	STP.B201B2_AirBlowerS2_RunStat AT %IX51.3 : BOOL;	(*  ~ {LinkedWith:TIID^C6920 (EtherCAT)^ScadaRoom_KouplerUTP (EK1100)^ScadaRoom_KouplerFiber (EK1521)^BlowerHouse_2 (EK1501)^Term 30 (EL1809)^Channel 14^Input} *)
	STP.B201B3_AirBlowerS2_RunStat AT %IX51.4 : BOOL;	(*  ~ {LinkedWith:TIID^C6920 (EtherCAT)^ScadaRoom_KouplerUTP (EK1100)^ScadaRoom_KouplerFiber (EK1521)^BlowerHouse_2 (EK1501)^Term 30 (EL1809)^Channel 15^Input} *)
	STP.M200B1A_MixerR1_LocalRemoteStat AT %IX51.5 : BOOL;	(*  ~ {LinkedWith:TIID^C6920 (EtherCAT)^ScadaRoom_KouplerUTP (EK1100)^ScadaRoom_KouplerFiber (EK1521)^BlowerHouse_2 (EK1501)^Term 31 (EL1809)^Channel 1^Input} *)
	STP.M200B1B_MixerR1_LocalRemoteStat AT %IX51.6 : BOOL;	(*  ~ {LinkedWith:TIID^C6920 (EtherCAT)^ScadaRoom_KouplerUTP (EK1100)^ScadaRoom_KouplerFiber (EK1521)^BlowerHouse_2 (EK1501)^Term 31 (EL1809)^Channel 2^Input} *)
	STP.M200B1C_MixerR1_LocalRemoteStat AT %IX51.7 : BOOL;	(*  ~ {LinkedWith:TIID^C6920 (EtherCAT)^ScadaRoom_KouplerUTP (EK1100)^ScadaRoom_KouplerFiber (EK1521)^BlowerHouse_2 (EK1501)^Term 31 (EL1809)^Channel 3^Input} *)
	STP.M200B2A_MixerR2_LocalRemoteStat AT %IX52.0 : BOOL;	(*  ~ {LinkedWith:TIID^C6920 (EtherCAT)^ScadaRoom_KouplerUTP (EK1100)^ScadaRoom_KouplerFiber (EK1521)^BlowerHouse_2 (EK1501)^Term 31 (EL1809)^Channel 4^Input} *)
	STP.M200B2B_MixerR2_LocalRemoteStat AT %IX52.1 : BOOL;	(*  ~ {LinkedWith:TIID^C6920 (EtherCAT)^ScadaRoom_KouplerUTP (EK1100)^ScadaRoom_KouplerFiber (EK1521)^BlowerHouse_2 (EK1501)^Term 31 (EL1809)^Channel 5^Input} *)
	STP.M200B2C_MixerR2_LocalRemoteStat AT %IX52.2 : BOOL;	(*  ~ {LinkedWith:TIID^C6920 (EtherCAT)^ScadaRoom_KouplerUTP (EK1100)^ScadaRoom_KouplerFiber (EK1521)^BlowerHouse_2 (EK1501)^Term 31 (EL1809)^Channel 6^Input} *)
	STP.M200B3A_MixerR3_LocalRemoteStat AT %IX52.3 : BOOL;	(*  ~ {LinkedWith:TIID^C6920 (EtherCAT)^ScadaRoom_KouplerUTP (EK1100)^ScadaRoom_KouplerFiber (EK1521)^BlowerHouse_2 (EK1501)^Term 31 (EL1809)^Channel 7^Input} *)
	STP.M200B3B_MixerR3_LocalRemoteStat AT %IX52.4 : BOOL;	(*  ~ {LinkedWith:TIID^C6920 (EtherCAT)^ScadaRoom_KouplerUTP (EK1100)^ScadaRoom_KouplerFiber (EK1521)^BlowerHouse_2 (EK1501)^Term 31 (EL1809)^Channel 8^Input} *)
	STP.M200B3C_MixerR3_LocalRemoteStat AT %IX52.5 : BOOL;	(*  ~ {LinkedWith:TIID^C6920 (EtherCAT)^ScadaRoom_KouplerUTP (EK1100)^ScadaRoom_KouplerFiber (EK1521)^BlowerHouse_2 (EK1501)^Term 31 (EL1809)^Channel 9^Input} *)
	STP.M200B4A_MixerR4_LocalRemoteStat AT %IX52.6 : BOOL;	(*  ~ {LinkedWith:TIID^C6920 (EtherCAT)^ScadaRoom_KouplerUTP (EK1100)^ScadaRoom_KouplerFiber (EK1521)^BlowerHouse_2 (EK1501)^Term 31 (EL1809)^Channel 10^Input} *)
	STP.M200B4B_MixerR4_LocalRemoteStat AT %IX52.7 : BOOL;	(*  ~ {LinkedWith:TIID^C6920 (EtherCAT)^ScadaRoom_KouplerUTP (EK1100)^ScadaRoom_KouplerFiber (EK1521)^BlowerHouse_2 (EK1501)^Term 31 (EL1809)^Channel 11^Input} *)
	STP.M200B4C_MixerR4_LocalRemoteStat AT %IX53.0 : BOOL;	(*  ~ {LinkedWith:TIID^C6920 (EtherCAT)^ScadaRoom_KouplerUTP (EK1100)^ScadaRoom_KouplerFiber (EK1521)^BlowerHouse_2 (EK1501)^Term 31 (EL1809)^Channel 12^Input} *)
	STP.B201B1_AirBlowerS2_LocalRemoteStat AT %IX53.1 : BOOL;	(*  ~ {LinkedWith:TIID^C6920 (EtherCAT)^ScadaRoom_KouplerUTP (EK1100)^ScadaRoom_KouplerFiber (EK1521)^BlowerHouse_2 (EK1501)^Term 32 (EL1809)^Channel 1^Input} *)
	STP.B201B2_AirBlowerS2_LocalRemoteStat AT %IX53.2 : BOOL;	(*  ~ {LinkedWith:TIID^C6920 (EtherCAT)^ScadaRoom_KouplerUTP (EK1100)^ScadaRoom_KouplerFiber (EK1521)^BlowerHouse_2 (EK1501)^Term 32 (EL1809)^Channel 2^Input} *)
	STP.B201B3_AirBlowerS2_LocalRemoteStat AT %IX53.3 : BOOL;	(*  ~ {LinkedWith:TIID^C6920 (EtherCAT)^ScadaRoom_KouplerUTP (EK1100)^ScadaRoom_KouplerFiber (EK1521)^BlowerHouse_2 (EK1501)^Term 32 (EL1809)^Channel 3^Input} *)
	STP.XV261B_DecanterR1_LocalRemoteStat AT %IX53.4 : BOOL;	(*  ~ {LinkedWith:TIID^C6920 (EtherCAT)^ScadaRoom_KouplerUTP (EK1100)^ScadaRoom_KouplerFiber (EK1521)^BlowerHouse_2 (EK1501)^Term 32 (EL1809)^Channel 4^Input} *)
	STP.XV262B_DecanterR2_LocalRemoteStat AT %IX53.5 : BOOL;	(*  ~ {LinkedWith:TIID^C6920 (EtherCAT)^ScadaRoom_KouplerUTP (EK1100)^ScadaRoom_KouplerFiber (EK1521)^BlowerHouse_2 (EK1501)^Term 32 (EL1809)^Channel 5^Input} *)
	STP.XV263B_DecanterR3_LocalRemoteStat AT %IX53.6 : BOOL;	(*  ~ {LinkedWith:TIID^C6920 (EtherCAT)^ScadaRoom_KouplerUTP (EK1100)^ScadaRoom_KouplerFiber (EK1521)^BlowerHouse_2 (EK1501)^Term 32 (EL1809)^Channel 6^Input} *)
	STP.XV264B_DecanterR4_LocalRemoteStat AT %IX53.7 : BOOL;	(*  ~ {LinkedWith:TIID^C6920 (EtherCAT)^ScadaRoom_KouplerUTP (EK1100)^ScadaRoom_KouplerFiber (EK1521)^BlowerHouse_2 (EK1501)^Term 32 (EL1809)^Channel 7^Input} *)
	STP.P201B1_DesludgePumpS2_LocalRemoteStat AT %IX54.0 : BOOL;	(*  ~ {LinkedWith:TIID^C6920 (EtherCAT)^ScadaRoom_KouplerUTP (EK1100)^ScadaRoom_KouplerFiber (EK1521)^BlowerHouse_2 (EK1501)^Term 32 (EL1809)^Channel 8^Input} *)
	STP.P201B2_DesludgePumpS2_LocalRemoteStat AT %IX54.1 : BOOL;	(*  ~ {LinkedWith:TIID^C6920 (EtherCAT)^ScadaRoom_KouplerUTP (EK1100)^ScadaRoom_KouplerFiber (EK1521)^BlowerHouse_2 (EK1501)^Term 32 (EL1809)^Channel 9^Input} *)
	STP.P201B1_DesludgePumpS2_RunStat AT %IX54.2 : BOOL;	(*  ~ {LinkedWith:TIID^C6920 (EtherCAT)^ScadaRoom_KouplerUTP (EK1100)^ScadaRoom_KouplerFiber (EK1521)^BlowerHouse_2 (EK1501)^Term 32 (EL1809)^Channel 10^Input} *)
	STP.P201B2_DesludgePumpS2_RunStat AT %IX54.3 : BOOL;	(*  ~ {LinkedWith:TIID^C6920 (EtherCAT)^ScadaRoom_KouplerUTP (EK1100)^ScadaRoom_KouplerFiber (EK1521)^BlowerHouse_2 (EK1501)^Term 32 (EL1809)^Channel 11^Input} *)
	STP.M200B1A_MixerR1_OverloadStat AT %IX54.4 : BOOL;	(*  ~ {LinkedWith:TIID^C6920 (EtherCAT)^ScadaRoom_KouplerUTP (EK1100)^ScadaRoom_KouplerFiber (EK1521)^BlowerHouse_2 (EK1501)^Term 33 (EL1809)^Channel 1^Input} *)
	STP.M200B1A_MixerR1_IncompleteStat AT %IX54.5 : BOOL;	(*  ~ {LinkedWith:TIID^C6920 (EtherCAT)^ScadaRoom_KouplerUTP (EK1100)^ScadaRoom_KouplerFiber (EK1521)^BlowerHouse_2 (EK1501)^Term 33 (EL1809)^Channel 2^Input} *)
	STP.M200B1B_MixerR1_OverloadStat AT %IX54.6 : BOOL;	(*  ~ {LinkedWith:TIID^C6920 (EtherCAT)^ScadaRoom_KouplerUTP (EK1100)^ScadaRoom_KouplerFiber (EK1521)^BlowerHouse_2 (EK1501)^Term 33 (EL1809)^Channel 3^Input} *)
	STP.M200B1B_MixerR1_IncompleteStat AT %IX54.7 : BOOL;	(*  ~ {LinkedWith:TIID^C6920 (EtherCAT)^ScadaRoom_KouplerUTP (EK1100)^ScadaRoom_KouplerFiber (EK1521)^BlowerHouse_2 (EK1501)^Term 33 (EL1809)^Channel 4^Input} *)
	STP.M200B1C_MixerR1_OverloadStat AT %IX55.0 : BOOL;	(*  ~ {LinkedWith:TIID^C6920 (EtherCAT)^ScadaRoom_KouplerUTP (EK1100)^ScadaRoom_KouplerFiber (EK1521)^BlowerHouse_2 (EK1501)^Term 33 (EL1809)^Channel 5^Input} *)
	STP.M200B1C_MixerR1_IncompleteStat AT %IX55.1 : BOOL;	(*  ~ {LinkedWith:TIID^C6920 (EtherCAT)^ScadaRoom_KouplerUTP (EK1100)^ScadaRoom_KouplerFiber (EK1521)^BlowerHouse_2 (EK1501)^Term 33 (EL1809)^Channel 6^Input} *)
	STP.M200B2A_MixerR2_OverloadStat AT %IX55.2 : BOOL;	(*  ~ {LinkedWith:TIID^C6920 (EtherCAT)^ScadaRoom_KouplerUTP (EK1100)^ScadaRoom_KouplerFiber (EK1521)^BlowerHouse_2 (EK1501)^Term 33 (EL1809)^Channel 7^Input} *)
	STP.M200B2A_MixerR2_IncompleteStat AT %IX55.3 : BOOL;	(*  ~ {LinkedWith:TIID^C6920 (EtherCAT)^ScadaRoom_KouplerUTP (EK1100)^ScadaRoom_KouplerFiber (EK1521)^BlowerHouse_2 (EK1501)^Term 33 (EL1809)^Channel 8^Input} *)
	STP.M200B2B_MixerR2_OverloadStat AT %IX55.4 : BOOL;	(*  ~ {LinkedWith:TIID^C6920 (EtherCAT)^ScadaRoom_KouplerUTP (EK1100)^ScadaRoom_KouplerFiber (EK1521)^BlowerHouse_2 (EK1501)^Term 33 (EL1809)^Channel 9^Input} *)
	STP.M200B2B_MixerR2_IncompleteStat AT %IX55.5 : BOOL;	(*  ~ {LinkedWith:TIID^C6920 (EtherCAT)^ScadaRoom_KouplerUTP (EK1100)^ScadaRoom_KouplerFiber (EK1521)^BlowerHouse_2 (EK1501)^Term 33 (EL1809)^Channel 10^Input} *)
	STP.M200B2C_MixerR2_OverloadStat AT %IX55.6 : BOOL;	(*  ~ {LinkedWith:TIID^C6920 (EtherCAT)^ScadaRoom_KouplerUTP (EK1100)^ScadaRoom_KouplerFiber (EK1521)^BlowerHouse_2 (EK1501)^Term 33 (EL1809)^Channel 11^Input} *)
	STP.M200B2C_MixerR2_IncompleteStat AT %IX55.7 : BOOL;	(*  ~ {LinkedWith:TIID^C6920 (EtherCAT)^ScadaRoom_KouplerUTP (EK1100)^ScadaRoom_KouplerFiber (EK1521)^BlowerHouse_2 (EK1501)^Term 33 (EL1809)^Channel 12^Input} *)
	STP.M200B3A_MixerR3_OverloadStat AT %IX56.0 : BOOL;	(*  ~ {LinkedWith:TIID^C6920 (EtherCAT)^ScadaRoom_KouplerUTP (EK1100)^ScadaRoom_KouplerFiber (EK1521)^BlowerHouse_2 (EK1501)^Term 33 (EL1809)^Channel 13^Input} *)
	STP.M200B3A_MixerR2_IncompleteStat AT %IX56.1 : BOOL;	(*  ~ {LinkedWith:TIID^C6920 (EtherCAT)^ScadaRoom_KouplerUTP (EK1100)^ScadaRoom_KouplerFiber (EK1521)^BlowerHouse_2 (EK1501)^Term 33 (EL1809)^Channel 14^Input} *)
	STP.M200B3B_MixerR3_OverloadStat AT %IX56.2 : BOOL;	(*  ~ {LinkedWith:TIID^C6920 (EtherCAT)^ScadaRoom_KouplerUTP (EK1100)^ScadaRoom_KouplerFiber (EK1521)^BlowerHouse_2 (EK1501)^Term 33 (EL1809)^Channel 15^Input} *)
	STP.M200B3B_MixerR3_IncompleteStat AT %IX56.3 : BOOL;	(*  ~ {LinkedWith:TIID^C6920 (EtherCAT)^ScadaRoom_KouplerUTP (EK1100)^ScadaRoom_KouplerFiber (EK1521)^BlowerHouse_2 (EK1501)^Term 33 (EL1809)^Channel 16^Input} *)
	STP.M200B3C_MixerR3_OverloadStat AT %IX56.4 : BOOL;	(*  ~ {LinkedWith:TIID^C6920 (EtherCAT)^ScadaRoom_KouplerUTP (EK1100)^ScadaRoom_KouplerFiber (EK1521)^BlowerHouse_2 (EK1501)^Term 34 (EL1809)^Channel 1^Input} *)
	STP.M200B3C_MixerR3_IncompleteStat AT %IX56.5 : BOOL;	(*  ~ {LinkedWith:TIID^C6920 (EtherCAT)^ScadaRoom_KouplerUTP (EK1100)^ScadaRoom_KouplerFiber (EK1521)^BlowerHouse_2 (EK1501)^Term 34 (EL1809)^Channel 2^Input} *)
	STP.M200B4A_MixerR4_OverloadStat AT %IX56.6 : BOOL;	(*  ~ {LinkedWith:TIID^C6920 (EtherCAT)^ScadaRoom_KouplerUTP (EK1100)^ScadaRoom_KouplerFiber (EK1521)^BlowerHouse_2 (EK1501)^Term 34 (EL1809)^Channel 3^Input} *)
	STP.M200B4A_MixerR4_IncompleteStat AT %IX56.7 : BOOL;	(*  ~ {LinkedWith:TIID^C6920 (EtherCAT)^ScadaRoom_KouplerUTP (EK1100)^ScadaRoom_KouplerFiber (EK1521)^BlowerHouse_2 (EK1501)^Term 34 (EL1809)^Channel 4^Input} *)
	STP.M200B4B_MixerR4_OverloadStat AT %IX257.0 : BOOL;	(*  ~ {LinkedWith:TIID^C6920 (EtherCAT)^ScadaRoom_KouplerUTP (EK1100)^ScadaRoom_KouplerFiber (EK1521)^BlowerHouse_2 (EK1501)^Term 34 (EL1809)^Channel 5^Input} *)
	STP.M200B4B_MixerR4_IncompleteStat AT %IX57.0 : BOOL;	(*  ~ {LinkedWith:TIID^C6920 (EtherCAT)^ScadaRoom_KouplerUTP (EK1100)^ScadaRoom_KouplerFiber (EK1521)^BlowerHouse_2 (EK1501)^Term 34 (EL1809)^Channel 6^Input} *)
	STP.M200B4C_MixerR4_OverloadStat AT %IX57.1 : BOOL;	(*  ~ {LinkedWith:TIID^C6920 (EtherCAT)^ScadaRoom_KouplerUTP (EK1100)^ScadaRoom_KouplerFiber (EK1521)^BlowerHouse_2 (EK1501)^Term 34 (EL1809)^Channel 7^Input} *)
	STP.M200B4C_MixerR4_IncompleteStat AT %IX57.2 : BOOL;	(*  ~ {LinkedWith:TIID^C6920 (EtherCAT)^ScadaRoom_KouplerUTP (EK1100)^ScadaRoom_KouplerFiber (EK1521)^BlowerHouse_2 (EK1501)^Term 34 (EL1809)^Channel 8^Input} *)
	STP.B201B1_AirBlowerS2_OverloadStat AT %IX57.3 : BOOL;	(*  ~ {LinkedWith:TIID^C6920 (EtherCAT)^ScadaRoom_KouplerUTP (EK1100)^ScadaRoom_KouplerFiber (EK1521)^BlowerHouse_2 (EK1501)^Term 34 (EL1809)^Channel 9^Input} *)
	STP.B201B1_AirBlowerS2_IncompleteStat AT %IX57.4 : BOOL;	(*  ~ {LinkedWith:TIID^C6920 (EtherCAT)^ScadaRoom_KouplerUTP (EK1100)^ScadaRoom_KouplerFiber (EK1521)^BlowerHouse_2 (EK1501)^Term 34 (EL1809)^Channel 10^Input} *)
	STP.B201B2_AirBlowerS2_OverloadStat AT %IX57.5 : BOOL;	(*  ~ {LinkedWith:TIID^C6920 (EtherCAT)^ScadaRoom_KouplerUTP (EK1100)^ScadaRoom_KouplerFiber (EK1521)^BlowerHouse_2 (EK1501)^Term 34 (EL1809)^Channel 11^Input} *)
	STP.B201B2_AirBlowerS2_IncompleteStat AT %IX57.6 : BOOL;	(*  ~ {LinkedWith:TIID^C6920 (EtherCAT)^ScadaRoom_KouplerUTP (EK1100)^ScadaRoom_KouplerFiber (EK1521)^BlowerHouse_2 (EK1501)^Term 34 (EL1809)^Channel 12^Input} *)
	STP.B201B3_AirBlowerS2_OverloadStat AT %IX57.7 : BOOL;	(*  ~ {LinkedWith:TIID^C6920 (EtherCAT)^ScadaRoom_KouplerUTP (EK1100)^ScadaRoom_KouplerFiber (EK1521)^BlowerHouse_2 (EK1501)^Term 34 (EL1809)^Channel 13^Input} *)
	STP.B201B3_AirBlowerS2_IncompleteStat AT %IX58.0 : BOOL;	(*  ~ {LinkedWith:TIID^C6920 (EtherCAT)^ScadaRoom_KouplerUTP (EK1100)^ScadaRoom_KouplerFiber (EK1521)^BlowerHouse_2 (EK1501)^Term 34 (EL1809)^Channel 14^Input} *)
	STP.P201B1_DesludgePumpS2_OverloadStat AT %IX58.1 : BOOL;	(*  ~ {LinkedWith:TIID^C6920 (EtherCAT)^ScadaRoom_KouplerUTP (EK1100)^ScadaRoom_KouplerFiber (EK1521)^BlowerHouse_2 (EK1501)^Term 34 (EL1809)^Channel 15^Input} *)
	STP.P201B2_DesludgePumpS2_OverloadStat AT %IX58.2 : BOOL;	(*  ~ {LinkedWith:TIID^C6920 (EtherCAT)^ScadaRoom_KouplerUTP (EK1100)^ScadaRoom_KouplerFiber (EK1521)^BlowerHouse_2 (EK1501)^Term 34 (EL1809)^Channel 16^Input} *)
	STP.M200B1A_MixerR1_EStopStat AT %IX58.3 : BOOL;	(*  ~ {LinkedWith:TIID^C6920 (EtherCAT)^ScadaRoom_KouplerUTP (EK1100)^ScadaRoom_KouplerFiber (EK1521)^BlowerHouse_2 (EK1501)^Term 35 (EL1809)^Channel 1^Input} *)
	STP.M200B1B_MixerR1_EStopStat AT %IX58.4 : BOOL;	(*  ~ {LinkedWith:TIID^C6920 (EtherCAT)^ScadaRoom_KouplerUTP (EK1100)^ScadaRoom_KouplerFiber (EK1521)^BlowerHouse_2 (EK1501)^Term 35 (EL1809)^Channel 2^Input} *)
	STP.M200B1C_MixerR1_EStopStat AT %IX58.5 : BOOL;	(*  ~ {LinkedWith:TIID^C6920 (EtherCAT)^ScadaRoom_KouplerUTP (EK1100)^ScadaRoom_KouplerFiber (EK1521)^BlowerHouse_2 (EK1501)^Term 35 (EL1809)^Channel 3^Input} *)
	STP.M200B2A_MixerR2_EStopStat AT %IX58.6 : BOOL;	(*  ~ {LinkedWith:TIID^C6920 (EtherCAT)^ScadaRoom_KouplerUTP (EK1100)^ScadaRoom_KouplerFiber (EK1521)^BlowerHouse_2 (EK1501)^Term 35 (EL1809)^Channel 4^Input} *)
	STP.M200B2B_MixerR2_EStopStat AT %IX58.7 : BOOL;	(*  ~ {LinkedWith:TIID^C6920 (EtherCAT)^ScadaRoom_KouplerUTP (EK1100)^ScadaRoom_KouplerFiber (EK1521)^BlowerHouse_2 (EK1501)^Term 35 (EL1809)^Channel 5^Input} *)
	STP.M200B2C_MixerR2_EStopStat AT %IX59.0 : BOOL;	(*  ~ {LinkedWith:TIID^C6920 (EtherCAT)^ScadaRoom_KouplerUTP (EK1100)^ScadaRoom_KouplerFiber (EK1521)^BlowerHouse_2 (EK1501)^Term 35 (EL1809)^Channel 6^Input} *)
	STP.M200B3A_MixerR3_EStopStat AT %IX59.1 : BOOL;	(*  ~ {LinkedWith:TIID^C6920 (EtherCAT)^ScadaRoom_KouplerUTP (EK1100)^ScadaRoom_KouplerFiber (EK1521)^BlowerHouse_2 (EK1501)^Term 35 (EL1809)^Channel 7^Input} *)
	STP.M200B3B_MixerR3_EStopStat AT %IX59.2 : BOOL;	(*  ~ {LinkedWith:TIID^C6920 (EtherCAT)^ScadaRoom_KouplerUTP (EK1100)^ScadaRoom_KouplerFiber (EK1521)^BlowerHouse_2 (EK1501)^Term 35 (EL1809)^Channel 8^Input} *)
	STP.M200B3C_MixerR3_EStopStat AT %IX59.3 : BOOL;	(*  ~ {LinkedWith:TIID^C6920 (EtherCAT)^ScadaRoom_KouplerUTP (EK1100)^ScadaRoom_KouplerFiber (EK1521)^BlowerHouse_2 (EK1501)^Term 35 (EL1809)^Channel 9^Input} *)
	STP.M200B4A_MixerR4_EStopStat AT %IX59.4 : BOOL;	(*  ~ {LinkedWith:TIID^C6920 (EtherCAT)^ScadaRoom_KouplerUTP (EK1100)^ScadaRoom_KouplerFiber (EK1521)^BlowerHouse_2 (EK1501)^Term 35 (EL1809)^Channel 10^Input} *)
	STP.M200B4B_MixerR4_EStopStat AT %IX59.5 : BOOL;	(*  ~ {LinkedWith:TIID^C6920 (EtherCAT)^ScadaRoom_KouplerUTP (EK1100)^ScadaRoom_KouplerFiber (EK1521)^BlowerHouse_2 (EK1501)^Term 35 (EL1809)^Channel 11^Input} *)
	STP.M200B4C_MixerR4_EStopStat AT %IX59.6 : BOOL;	(*  ~ {LinkedWith:TIID^C6920 (EtherCAT)^ScadaRoom_KouplerUTP (EK1100)^ScadaRoom_KouplerFiber (EK1521)^BlowerHouse_2 (EK1501)^Term 35 (EL1809)^Channel 12^Input} *)
	STP.B201B1_AirBlowerS2_EStopStat AT %IX59.7 : BOOL;	(*  ~ {LinkedWith:TIID^C6920 (EtherCAT)^ScadaRoom_KouplerUTP (EK1100)^ScadaRoom_KouplerFiber (EK1521)^BlowerHouse_2 (EK1501)^Term 36 (EL1809)^Channel 1^Input} *)
	STP.B201B2_AirBlowerS2_EStopStat AT %IX60.0 : BOOL;	(*  ~ {LinkedWith:TIID^C6920 (EtherCAT)^ScadaRoom_KouplerUTP (EK1100)^ScadaRoom_KouplerFiber (EK1521)^BlowerHouse_2 (EK1501)^Term 36 (EL1809)^Channel 2^Input} *)
	STP.B201B3_AirBlowerS2_EStopStat AT %IX60.1 : BOOL;	(*  ~ {LinkedWith:TIID^C6920 (EtherCAT)^ScadaRoom_KouplerUTP (EK1100)^ScadaRoom_KouplerFiber (EK1521)^BlowerHouse_2 (EK1501)^Term 36 (EL1809)^Channel 3^Input} *)
	STP.XV261B_DecanterR1_EStopStat AT %IX60.2 : BOOL;	(*  ~ {LinkedWith:TIID^C6920 (EtherCAT)^ScadaRoom_KouplerUTP (EK1100)^ScadaRoom_KouplerFiber (EK1521)^BlowerHouse_2 (EK1501)^Term 36 (EL1809)^Channel 4^Input} *)
	STP.XV262B_DecanterR2_EStopStat AT %IX60.3 : BOOL;	(*  ~ {LinkedWith:TIID^C6920 (EtherCAT)^ScadaRoom_KouplerUTP (EK1100)^ScadaRoom_KouplerFiber (EK1521)^BlowerHouse_2 (EK1501)^Term 36 (EL1809)^Channel 5^Input} *)
	STP.XV263B_DecanterR3_EStopStat AT %IX60.4 : BOOL;	(*  ~ {LinkedWith:TIID^C6920 (EtherCAT)^ScadaRoom_KouplerUTP (EK1100)^ScadaRoom_KouplerFiber (EK1521)^BlowerHouse_2 (EK1501)^Term 36 (EL1809)^Channel 6^Input} *)
	STP.XV264B_DecanterR4_EStopStat AT %IX60.5 : BOOL;	(*  ~ {LinkedWith:TIID^C6920 (EtherCAT)^ScadaRoom_KouplerUTP (EK1100)^ScadaRoom_KouplerFiber (EK1521)^BlowerHouse_2 (EK1501)^Term 36 (EL1809)^Channel 7^Input} *)
	STP.P201B1_DesludgePumpS2_EStopStat AT %IX60.6 : BOOL;	(*  ~ {LinkedWith:TIID^C6920 (EtherCAT)^ScadaRoom_KouplerUTP (EK1100)^ScadaRoom_KouplerFiber (EK1521)^BlowerHouse_2 (EK1501)^Term 36 (EL1809)^Channel 8^Input} *)
	STP.P201B2_DesludgePumpS2_EStopStat AT %IX60.7 : BOOL;	(*  ~ {LinkedWith:TIID^C6920 (EtherCAT)^ScadaRoom_KouplerUTP (EK1100)^ScadaRoom_KouplerFiber (EK1521)^BlowerHouse_2 (EK1501)^Term 36 (EL1809)^Channel 9^Input} *)
	STP.XV261B_DecanterR1_FwdStat AT %IX61.0 : BOOL;	(*  ~ {LinkedWith:TIID^C6920 (EtherCAT)^ScadaRoom_KouplerUTP (EK1100)^ScadaRoom_KouplerFiber (EK1521)^BlowerHouse_2 (EK1501)^Term 37 (EL1809)^Channel 1^Input} *)
	STP.XV262B_DecanterR2_FwdStat AT %IX61.1 : BOOL;	(*  ~ {LinkedWith:TIID^C6920 (EtherCAT)^ScadaRoom_KouplerUTP (EK1100)^ScadaRoom_KouplerFiber (EK1521)^BlowerHouse_2 (EK1501)^Term 37 (EL1809)^Channel 2^Input} *)
	STP.XV263B_DecanterR3_FwdStat AT %IX61.2 : BOOL;	(*  ~ {LinkedWith:TIID^C6920 (EtherCAT)^ScadaRoom_KouplerUTP (EK1100)^ScadaRoom_KouplerFiber (EK1521)^BlowerHouse_2 (EK1501)^Term 37 (EL1809)^Channel 3^Input} *)
	STP.XV264B_DecanterR4_FwdStat AT %IX61.3 : BOOL;	(*  ~ {LinkedWith:TIID^C6920 (EtherCAT)^ScadaRoom_KouplerUTP (EK1100)^ScadaRoom_KouplerFiber (EK1521)^BlowerHouse_2 (EK1501)^Term 37 (EL1809)^Channel 4^Input} *)
	STP.XV261B_DecanterR1_RvsStat AT %IX61.4 : BOOL;	(*  ~ {LinkedWith:TIID^C6920 (EtherCAT)^ScadaRoom_KouplerUTP (EK1100)^ScadaRoom_KouplerFiber (EK1521)^BlowerHouse_2 (EK1501)^Term 37 (EL1809)^Channel 5^Input} *)
	STP.XV262B_DecanterR2_RvsStat AT %IX61.5 : BOOL;	(*  ~ {LinkedWith:TIID^C6920 (EtherCAT)^ScadaRoom_KouplerUTP (EK1100)^ScadaRoom_KouplerFiber (EK1521)^BlowerHouse_2 (EK1501)^Term 37 (EL1809)^Channel 6^Input} *)
	STP.XV263B_DecanterR3_RvsStat AT %IX61.6 : BOOL;	(*  ~ {LinkedWith:TIID^C6920 (EtherCAT)^ScadaRoom_KouplerUTP (EK1100)^ScadaRoom_KouplerFiber (EK1521)^BlowerHouse_2 (EK1501)^Term 37 (EL1809)^Channel 7^Input} *)
	STP.XV264B_DecanterR4_RvsStat AT %IX61.7 : BOOL;	(*  ~ {LinkedWith:TIID^C6920 (EtherCAT)^ScadaRoom_KouplerUTP (EK1100)^ScadaRoom_KouplerFiber (EK1521)^BlowerHouse_2 (EK1501)^Term 37 (EL1809)^Channel 8^Input} *)
	STP.M200B1A_MixerR1_RunCmd AT %QX17.1 : BOOL;	(*  ~ {LinkedWith:TIID^C6920 (EtherCAT)^ScadaRoom_KouplerUTP (EK1100)^ScadaRoom_KouplerFiber (EK1521)^BlowerHouse_2 (EK1501)^Term 39 (EL2809)^Channel 1^Output} *)
	STP.M200B1B_MixerR1_RunCmd AT %QX17.2 : BOOL;	(*  ~ {LinkedWith:TIID^C6920 (EtherCAT)^ScadaRoom_KouplerUTP (EK1100)^ScadaRoom_KouplerFiber (EK1521)^BlowerHouse_2 (EK1501)^Term 39 (EL2809)^Channel 2^Output} *)
	STP.M200B1C_MixerR1_RunCmd AT %QX17.3 : BOOL;	(*  ~ {LinkedWith:TIID^C6920 (EtherCAT)^ScadaRoom_KouplerUTP (EK1100)^ScadaRoom_KouplerFiber (EK1521)^BlowerHouse_2 (EK1501)^Term 39 (EL2809)^Channel 3^Output} *)
	STP.M200B2A_MixerR2_RunCmd AT %QX17.4 : BOOL;	(*  ~ {LinkedWith:TIID^C6920 (EtherCAT)^ScadaRoom_KouplerUTP (EK1100)^ScadaRoom_KouplerFiber (EK1521)^BlowerHouse_2 (EK1501)^Term 39 (EL2809)^Channel 4^Output} *)
	STP.M200B2B_MixerR2_RunCmd AT %QX17.5 : BOOL;	(*  ~ {LinkedWith:TIID^C6920 (EtherCAT)^ScadaRoom_KouplerUTP (EK1100)^ScadaRoom_KouplerFiber (EK1521)^BlowerHouse_2 (EK1501)^Term 39 (EL2809)^Channel 5^Output} *)
	STP.M200B2C_MixerR2_RunCmd AT %QX17.6 : BOOL;	(*  ~ {LinkedWith:TIID^C6920 (EtherCAT)^ScadaRoom_KouplerUTP (EK1100)^ScadaRoom_KouplerFiber (EK1521)^BlowerHouse_2 (EK1501)^Term 39 (EL2809)^Channel 6^Output} *)
	STP.M200B3A_MixerR3_RunCmd AT %QX17.7 : BOOL;	(*  ~ {LinkedWith:TIID^C6920 (EtherCAT)^ScadaRoom_KouplerUTP (EK1100)^ScadaRoom_KouplerFiber (EK1521)^BlowerHouse_2 (EK1501)^Term 39 (EL2809)^Channel 7^Output} *)
	STP.M200B3B_MixerR3_RunCmd AT %QX18.0 : BOOL;	(*  ~ {LinkedWith:TIID^C6920 (EtherCAT)^ScadaRoom_KouplerUTP (EK1100)^ScadaRoom_KouplerFiber (EK1521)^BlowerHouse_2 (EK1501)^Term 39 (EL2809)^Channel 8^Output} *)
	STP.M200B3C_MixerR3_RunCmd AT %QX18.1 : BOOL;	(*  ~ {LinkedWith:TIID^C6920 (EtherCAT)^ScadaRoom_KouplerUTP (EK1100)^ScadaRoom_KouplerFiber (EK1521)^BlowerHouse_2 (EK1501)^Term 39 (EL2809)^Channel 9^Output} *)
	STP.M200B4A_MixerR4_RunCmd AT %QX18.2 : BOOL;	(*  ~ {LinkedWith:TIID^C6920 (EtherCAT)^ScadaRoom_KouplerUTP (EK1100)^ScadaRoom_KouplerFiber (EK1521)^BlowerHouse_2 (EK1501)^Term 39 (EL2809)^Channel 10^Output} *)
	STP.M200B4B_MixerR4_RunCmd AT %QX18.3 : BOOL;	(*  ~ {LinkedWith:TIID^C6920 (EtherCAT)^ScadaRoom_KouplerUTP (EK1100)^ScadaRoom_KouplerFiber (EK1521)^BlowerHouse_2 (EK1501)^Term 39 (EL2809)^Channel 11^Output} *)
	STP.M200B4C_MixerR4_RunCmd AT %QX18.4 : BOOL;	(*  ~ {LinkedWith:TIID^C6920 (EtherCAT)^ScadaRoom_KouplerUTP (EK1100)^ScadaRoom_KouplerFiber (EK1521)^BlowerHouse_2 (EK1501)^Term 39 (EL2809)^Channel 12^Output} *)
	STP.XV261B_DecanterR1_FwdCmd AT %QX18.5 : BOOL;	(*  ~ {LinkedWith:TIID^C6920 (EtherCAT)^ScadaRoom_KouplerUTP (EK1100)^ScadaRoom_KouplerFiber (EK1521)^BlowerHouse_2 (EK1501)^Term 40 (EL2809)^Channel 1^Output} *)
	STP.XV262B_DecanterR2_FwdCmd AT %QX18.6 : BOOL;	(*  ~ {LinkedWith:TIID^C6920 (EtherCAT)^ScadaRoom_KouplerUTP (EK1100)^ScadaRoom_KouplerFiber (EK1521)^BlowerHouse_2 (EK1501)^Term 40 (EL2809)^Channel 2^Output} *)
	STP.XV263B_DecanterR3_FwdCmd AT %QX18.7 : BOOL;	(*  ~ {LinkedWith:TIID^C6920 (EtherCAT)^ScadaRoom_KouplerUTP (EK1100)^ScadaRoom_KouplerFiber (EK1521)^BlowerHouse_2 (EK1501)^Term 40 (EL2809)^Channel 3^Output} *)
	STP.XV264B_DecanterR4_FwdCmd AT %QX19.0 : BOOL;	(*  ~ {LinkedWith:TIID^C6920 (EtherCAT)^ScadaRoom_KouplerUTP (EK1100)^ScadaRoom_KouplerFiber (EK1521)^BlowerHouse_2 (EK1501)^Term 40 (EL2809)^Channel 4^Output} *)
	STP.XV261B_DecanterR1_RvsCmd AT %QX19.1 : BOOL;	(*  ~ {LinkedWith:TIID^C6920 (EtherCAT)^ScadaRoom_KouplerUTP (EK1100)^ScadaRoom_KouplerFiber (EK1521)^BlowerHouse_2 (EK1501)^Term 40 (EL2809)^Channel 5^Output} *)
	STP.XV262B_DecanterR2_RvsCmd AT %QX19.2 : BOOL;	(*  ~ {LinkedWith:TIID^C6920 (EtherCAT)^ScadaRoom_KouplerUTP (EK1100)^ScadaRoom_KouplerFiber (EK1521)^BlowerHouse_2 (EK1501)^Term 40 (EL2809)^Channel 6^Output} *)
	STP.XV263B_DecanterR3_RvsCmd AT %QX19.3 : BOOL;	(*  ~ {LinkedWith:TIID^C6920 (EtherCAT)^ScadaRoom_KouplerUTP (EK1100)^ScadaRoom_KouplerFiber (EK1521)^BlowerHouse_2 (EK1501)^Term 40 (EL2809)^Channel 7^Output} *)
	STP.XV264B_DecanterR4_RvsCmd AT %QX19.4 : BOOL;	(*  ~ {LinkedWith:TIID^C6920 (EtherCAT)^ScadaRoom_KouplerUTP (EK1100)^ScadaRoom_KouplerFiber (EK1521)^BlowerHouse_2 (EK1501)^Term 40 (EL2809)^Channel 8^Output} *)
	STP.B201B1_AirBlowerS2_RunCmd AT %QX19.5 : BOOL;	(*  ~ {LinkedWith:TIID^C6920 (EtherCAT)^ScadaRoom_KouplerUTP (EK1100)^ScadaRoom_KouplerFiber (EK1521)^BlowerHouse_2 (EK1501)^Term 40 (EL2809)^Channel 9^Output} *)
	STP.B201B2_AirBlowerS2_RunCmd AT %QX19.6 : BOOL;	(*  ~ {LinkedWith:TIID^C6920 (EtherCAT)^ScadaRoom_KouplerUTP (EK1100)^ScadaRoom_KouplerFiber (EK1521)^BlowerHouse_2 (EK1501)^Term 40 (EL2809)^Channel 10^Output} *)
	STP.B201B3_AirBlowerS2_RunCmd AT %QX19.7 : BOOL;	(*  ~ {LinkedWith:TIID^C6920 (EtherCAT)^ScadaRoom_KouplerUTP (EK1100)^ScadaRoom_KouplerFiber (EK1521)^BlowerHouse_2 (EK1501)^Term 40 (EL2809)^Channel 11^Output} *)
	STP.P201B1_DesludgePumpS2_RunCmd AT %QX20.0 : BOOL;	(*  ~ {LinkedWith:TIID^C6920 (EtherCAT)^ScadaRoom_KouplerUTP (EK1100)^ScadaRoom_KouplerFiber (EK1521)^BlowerHouse_2 (EK1501)^Term 40 (EL2809)^Channel 12^Output} *)
	STP.P201B2_DesludgePumpS2_RunCmd AT %QX20.1 : BOOL;	(*  ~ {LinkedWith:TIID^C6920 (EtherCAT)^ScadaRoom_KouplerUTP (EK1100)^ScadaRoom_KouplerFiber (EK1521)^BlowerHouse_2 (EK1501)^Term 40 (EL2809)^Channel 13^Output} *)
	STP.LSH201A1_LevelSensorR1 AT %IX64.0 : BOOL;	(*  ~ {LinkedWith:TIID^C6920 (EtherCAT)^ScadaRoom_KouplerUTP (EK1100)^ScadaRoom_KouplerFiber (EK1521)^SBR_1 (EK1501)^Term 57 (EL1809)^Channel 1^Input} *)
	STP.LSH201A2_LevelSensorR2 AT %IX64.1 : BOOL;	(*  ~ {LinkedWith:TIID^C6920 (EtherCAT)^ScadaRoom_KouplerUTP (EK1100)^ScadaRoom_KouplerFiber (EK1521)^SBR_1 (EK1501)^Term 57 (EL1809)^Channel 2^Input} *)
	STP.LSH201A3_LevelSensorR3 AT %IX64.2 : BOOL;	(*  ~ {LinkedWith:TIID^C6920 (EtherCAT)^ScadaRoom_KouplerUTP (EK1100)^ScadaRoom_KouplerFiber (EK1521)^SBR_1 (EK1501)^Term 57 (EL1809)^Channel 3^Input} *)
	STP.LSH201A4_LevelSensorR4 AT %IX64.3 : BOOL;	(*  ~ {LinkedWith:TIID^C6920 (EtherCAT)^ScadaRoom_KouplerUTP (EK1100)^ScadaRoom_KouplerFiber (EK1521)^SBR_1 (EK1501)^Term 57 (EL1809)^Channel 4^Input} *)
	STP.OPR1A_ReactorStatus AT %IX64.4 : BOOL;	(*  ~ {LinkedWith:TIID^C6920 (EtherCAT)^ScadaRoom_KouplerUTP (EK1100)^ScadaRoom_KouplerFiber (EK1521)^SBR_1 (EK1501)^Term 57 (EL1809)^Channel 5^Input} *)
	STP.OPR2A_ReactorStatus AT %IX64.5 : BOOL;	(*  ~ {LinkedWith:TIID^C6920 (EtherCAT)^ScadaRoom_KouplerUTP (EK1100)^ScadaRoom_KouplerFiber (EK1521)^SBR_1 (EK1501)^Term 57 (EL1809)^Channel 6^Input} *)
	STP.OPR3A_ReactorStatus AT %IX64.6 : BOOL;	(*  ~ {LinkedWith:TIID^C6920 (EtherCAT)^ScadaRoom_KouplerUTP (EK1100)^ScadaRoom_KouplerFiber (EK1521)^SBR_1 (EK1501)^Term 57 (EL1809)^Channel 7^Input} *)
	STP.OPR4A_ReactorStatus AT %IX64.7 : BOOL;	(*  ~ {LinkedWith:TIID^C6920 (EtherCAT)^ScadaRoom_KouplerUTP (EK1100)^ScadaRoom_KouplerFiber (EK1521)^SBR_1 (EK1501)^Term 57 (EL1809)^Channel 8^Input} *)
	STP.DP04_DoorPanelStatus AT %IX65.0 : BOOL;	(*  ~ {LinkedWith:TIID^C6920 (EtherCAT)^ScadaRoom_KouplerUTP (EK1100)^ScadaRoom_KouplerFiber (EK1521)^SBR_1 (EK1501)^Term 57 (EL1809)^Channel 9^Input} *)
	STP.TMT04_FanStatus AT %IX65.1 : BOOL;	(*  ~ {LinkedWith:TIID^C6920 (EtherCAT)^ScadaRoom_KouplerUTP (EK1100)^ScadaRoom_KouplerFiber (EK1521)^SBR_1 (EK1501)^Term 57 (EL1809)^Channel 10^Input} *)
	STP.HR201A1_DecantHighLevelR1 AT %IX65.2 : BOOL;	(*  ~ {LinkedWith:TIID^C6920 (EtherCAT)^ScadaRoom_KouplerUTP (EK1100)^ScadaRoom_KouplerFiber (EK1521)^SBR_1 (EK1501)^Term 58 (EL1809)^Channel 1^Input} *)
	STP.LR201A1_DecantLowLevelR1 AT %IX65.3 : BOOL;	(*  ~ {LinkedWith:TIID^C6920 (EtherCAT)^ScadaRoom_KouplerUTP (EK1100)^ScadaRoom_KouplerFiber (EK1521)^SBR_1 (EK1501)^Term 58 (EL1809)^Channel 2^Input} *)
	STP.HR201A2_DecantHighLevelR2 AT %IX65.4 : BOOL;	(*  ~ {LinkedWith:TIID^C6920 (EtherCAT)^ScadaRoom_KouplerUTP (EK1100)^ScadaRoom_KouplerFiber (EK1521)^SBR_1 (EK1501)^Term 58 (EL1809)^Channel 3^Input} *)
	STP.LR201A2_DecantLowLevelR2 AT %IX65.5 : BOOL;	(*  ~ {LinkedWith:TIID^C6920 (EtherCAT)^ScadaRoom_KouplerUTP (EK1100)^ScadaRoom_KouplerFiber (EK1521)^SBR_1 (EK1501)^Term 58 (EL1809)^Channel 4^Input} *)
	STP.HR201A3_DecantHighLevelR3 AT %IX65.6 : BOOL;	(*  ~ {LinkedWith:TIID^C6920 (EtherCAT)^ScadaRoom_KouplerUTP (EK1100)^ScadaRoom_KouplerFiber (EK1521)^SBR_1 (EK1501)^Term 58 (EL1809)^Channel 5^Input} *)
	STP.LR201A3_DecantLowLevelR3 AT %IX65.7 : BOOL;	(*  ~ {LinkedWith:TIID^C6920 (EtherCAT)^ScadaRoom_KouplerUTP (EK1100)^ScadaRoom_KouplerFiber (EK1521)^SBR_1 (EK1501)^Term 58 (EL1809)^Channel 6^Input} *)
	STP.HR201A4_DecantHighLevelR4 AT %IX66.0 : BOOL;	(*  ~ {LinkedWith:TIID^C6920 (EtherCAT)^ScadaRoom_KouplerUTP (EK1100)^ScadaRoom_KouplerFiber (EK1521)^SBR_1 (EK1501)^Term 58 (EL1809)^Channel 7^Input} *)
	STP.LR201A4_DecantLowLevelR4 AT %IX66.1 : BOOL;	(*  ~ {LinkedWith:TIID^C6920 (EtherCAT)^ScadaRoom_KouplerUTP (EK1100)^ScadaRoom_KouplerFiber (EK1521)^SBR_1 (EK1501)^Term 58 (EL1809)^Channel 8^Input} *)
	STP.XV205A_SBRValveR1_OpenStat AT %IX66.2 : BOOL;	(*  ~ {LinkedWith:TIID^C6920 (EtherCAT)^ScadaRoom_KouplerUTP (EK1100)^ScadaRoom_KouplerFiber (EK1521)^SBR_1 (EK1501)^Term 59 (EL1809)^Channel 1^Input} *)
	STP.XV206A_SBRValveR2_OpenStat AT %IX66.3 : BOOL;	(*  ~ {LinkedWith:TIID^C6920 (EtherCAT)^ScadaRoom_KouplerUTP (EK1100)^ScadaRoom_KouplerFiber (EK1521)^SBR_1 (EK1501)^Term 59 (EL1809)^Channel 2^Input} *)
	STP.XV207A_SBRValveR3_OpenStat AT %IX66.4 : BOOL;	(*  ~ {LinkedWith:TIID^C6920 (EtherCAT)^ScadaRoom_KouplerUTP (EK1100)^ScadaRoom_KouplerFiber (EK1521)^SBR_1 (EK1501)^Term 59 (EL1809)^Channel 3^Input} *)
	STP.XV208A_SBRValveR4_OpenStat AT %IX66.5 : BOOL;	(*  ~ {LinkedWith:TIID^C6920 (EtherCAT)^ScadaRoom_KouplerUTP (EK1100)^ScadaRoom_KouplerFiber (EK1521)^SBR_1 (EK1501)^Term 59 (EL1809)^Channel 4^Input} *)
	STP.XV201A_AirBlowerValveR1_OpenStat AT %IX66.6 : BOOL;	(*  ~ {LinkedWith:TIID^C6920 (EtherCAT)^ScadaRoom_KouplerUTP (EK1100)^ScadaRoom_KouplerFiber (EK1521)^SBR_1 (EK1501)^Term 59 (EL1809)^Channel 5^Input} *)
	STP.XV202A_AirBlowerValveR2_OpenStat AT %IX66.7 : BOOL;	(*  ~ {LinkedWith:TIID^C6920 (EtherCAT)^ScadaRoom_KouplerUTP (EK1100)^ScadaRoom_KouplerFiber (EK1521)^SBR_1 (EK1501)^Term 59 (EL1809)^Channel 6^Input} *)
	STP.XV203A_AirBlowerValveR3_OpenStat AT %IX67.0 : BOOL;	(*  ~ {LinkedWith:TIID^C6920 (EtherCAT)^ScadaRoom_KouplerUTP (EK1100)^ScadaRoom_KouplerFiber (EK1521)^SBR_1 (EK1501)^Term 59 (EL1809)^Channel 7^Input} *)
	STP.XV204A_AirBlowerValveR4_OpenStat AT %IX68.1 : BOOL;	(*  ~ {LinkedWith:TIID^C6920 (EtherCAT)^ScadaRoom_KouplerUTP (EK1100)^ScadaRoom_KouplerFiber (EK1521)^SBR_1 (EK1501)^Term 59 (EL1809)^Channel 8^Input} *)
	STP.XV221A_LimeValveR1_OpenStat AT %IX67.1 : BOOL;	(*  ~ {LinkedWith:TIID^C6920 (EtherCAT)^ScadaRoom_KouplerUTP (EK1100)^ScadaRoom_KouplerFiber (EK1521)^SBR_1 (EK1501)^Term 59 (EL1809)^Channel 9^Input} *)
	STP.XV222A_LimeValveR2_OpenStat AT %IX67.2 : BOOL;	(*  ~ {LinkedWith:TIID^C6920 (EtherCAT)^ScadaRoom_KouplerUTP (EK1100)^ScadaRoom_KouplerFiber (EK1521)^SBR_1 (EK1501)^Term 59 (EL1809)^Channel 10^Input} *)
	STP.XV223A_LimeValveR3_OpenStat AT %IX67.3 : BOOL;	(*  ~ {LinkedWith:TIID^C6920 (EtherCAT)^ScadaRoom_KouplerUTP (EK1100)^ScadaRoom_KouplerFiber (EK1521)^SBR_1 (EK1501)^Term 59 (EL1809)^Channel 11^Input} *)
	STP.XV224A_LimeValveR4_OpenStat AT %IX67.4 : BOOL;	(*  ~ {LinkedWith:TIID^C6920 (EtherCAT)^ScadaRoom_KouplerUTP (EK1100)^ScadaRoom_KouplerFiber (EK1521)^SBR_1 (EK1501)^Term 59 (EL1809)^Channel 12^Input} *)
	STP.XV211A_AlumValveR1_OpenStat AT %IX67.5 : BOOL;	(*  ~ {LinkedWith:TIID^C6920 (EtherCAT)^ScadaRoom_KouplerUTP (EK1100)^ScadaRoom_KouplerFiber (EK1521)^SBR_1 (EK1501)^Term 59 (EL1809)^Channel 13^Input} *)
	STP.XV212A_AlumValveR2_OpenStat AT %IX67.6 : BOOL;	(*  ~ {LinkedWith:TIID^C6920 (EtherCAT)^ScadaRoom_KouplerUTP (EK1100)^ScadaRoom_KouplerFiber (EK1521)^SBR_1 (EK1501)^Term 59 (EL1809)^Channel 14^Input} *)
	STP.XV213A_AlumValveR3_OpenStat AT %IX67.7 : BOOL;	(*  ~ {LinkedWith:TIID^C6920 (EtherCAT)^ScadaRoom_KouplerUTP (EK1100)^ScadaRoom_KouplerFiber (EK1521)^SBR_1 (EK1501)^Term 59 (EL1809)^Channel 15^Input} *)
	STP.XV214A_AlumValveR4_OpenStat AT %IX68.0 : BOOL;	(*  ~ {LinkedWith:TIID^C6920 (EtherCAT)^ScadaRoom_KouplerUTP (EK1100)^ScadaRoom_KouplerFiber (EK1521)^SBR_1 (EK1501)^Term 59 (EL1809)^Channel 16^Input} *)
	STP.XV205A_SBRValveR1_CloseStat AT %IX68.2 : BOOL;	(*  ~ {LinkedWith:TIID^C6920 (EtherCAT)^ScadaRoom_KouplerUTP (EK1100)^ScadaRoom_KouplerFiber (EK1521)^SBR_1 (EK1501)^Term 60 (EL1809)^Channel 1^Input} *)
	STP.XV206A_SBRValveR2_CloseStat AT %IX68.3 : BOOL;	(*  ~ {LinkedWith:TIID^C6920 (EtherCAT)^ScadaRoom_KouplerUTP (EK1100)^ScadaRoom_KouplerFiber (EK1521)^SBR_1 (EK1501)^Term 60 (EL1809)^Channel 2^Input} *)
	STP.XV207A_SBRValveR3_CloseStat AT %IX68.4 : BOOL;	(*  ~ {LinkedWith:TIID^C6920 (EtherCAT)^ScadaRoom_KouplerUTP (EK1100)^ScadaRoom_KouplerFiber (EK1521)^SBR_1 (EK1501)^Term 60 (EL1809)^Channel 3^Input} *)
	STP.XV208A_SBRValveR4_CloseStat AT %IX68.5 : BOOL;	(*  ~ {LinkedWith:TIID^C6920 (EtherCAT)^ScadaRoom_KouplerUTP (EK1100)^ScadaRoom_KouplerFiber (EK1521)^SBR_1 (EK1501)^Term 60 (EL1809)^Channel 4^Input} *)
	STP.XV201A_AirBlowerValveR1_CloseStat AT %IX68.6 : BOOL;	(*  ~ {LinkedWith:TIID^C6920 (EtherCAT)^ScadaRoom_KouplerUTP (EK1100)^ScadaRoom_KouplerFiber (EK1521)^SBR_1 (EK1501)^Term 60 (EL1809)^Channel 5^Input} *)
	STP.XV202A_AirBlowerValveR2_CloseStat AT %IX68.7 : BOOL;	(*  ~ {LinkedWith:TIID^C6920 (EtherCAT)^ScadaRoom_KouplerUTP (EK1100)^ScadaRoom_KouplerFiber (EK1521)^SBR_1 (EK1501)^Term 60 (EL1809)^Channel 6^Input} *)
	STP.XV203A_AirBlowerValveR3_CloseStat AT %IX69.0 : BOOL;	(*  ~ {LinkedWith:TIID^C6920 (EtherCAT)^ScadaRoom_KouplerUTP (EK1100)^ScadaRoom_KouplerFiber (EK1521)^SBR_1 (EK1501)^Term 60 (EL1809)^Channel 7^Input} *)
	STP.XV204A_AirBlowerValveR4_CloseStat AT %IX69.1 : BOOL;	(*  ~ {LinkedWith:TIID^C6920 (EtherCAT)^ScadaRoom_KouplerUTP (EK1100)^ScadaRoom_KouplerFiber (EK1521)^SBR_1 (EK1501)^Term 60 (EL1809)^Channel 8^Input} *)
	STP.XV221A_LimeValveR1_CloseStat AT %IX69.2 : BOOL;	(*  ~ {LinkedWith:TIID^C6920 (EtherCAT)^ScadaRoom_KouplerUTP (EK1100)^ScadaRoom_KouplerFiber (EK1521)^SBR_1 (EK1501)^Term 60 (EL1809)^Channel 9^Input} *)
	STP.XV222A_LimeValveR2_CloseStat AT %IX69.3 : BOOL;	(*  ~ {LinkedWith:TIID^C6920 (EtherCAT)^ScadaRoom_KouplerUTP (EK1100)^ScadaRoom_KouplerFiber (EK1521)^SBR_1 (EK1501)^Term 60 (EL1809)^Channel 10^Input} *)
	STP.XV223A_LimeValveR3_CloseStat AT %IX69.4 : BOOL;	(*  ~ {LinkedWith:TIID^C6920 (EtherCAT)^ScadaRoom_KouplerUTP (EK1100)^ScadaRoom_KouplerFiber (EK1521)^SBR_1 (EK1501)^Term 60 (EL1809)^Channel 11^Input} *)
	STP.XV224A_LimeValveR4_CloseStat AT %IX69.5 : BOOL;	(*  ~ {LinkedWith:TIID^C6920 (EtherCAT)^ScadaRoom_KouplerUTP (EK1100)^ScadaRoom_KouplerFiber (EK1521)^SBR_1 (EK1501)^Term 60 (EL1809)^Channel 12^Input} *)
	STP.XV211A_AlumValveR1_CloseStat AT %IX69.6 : BOOL;	(*  ~ {LinkedWith:TIID^C6920 (EtherCAT)^ScadaRoom_KouplerUTP (EK1100)^ScadaRoom_KouplerFiber (EK1521)^SBR_1 (EK1501)^Term 60 (EL1809)^Channel 13^Input} *)
	STP.XV212A_AlumValveR2_CloseStat AT %IX69.7 : BOOL;	(*  ~ {LinkedWith:TIID^C6920 (EtherCAT)^ScadaRoom_KouplerUTP (EK1100)^ScadaRoom_KouplerFiber (EK1521)^SBR_1 (EK1501)^Term 60 (EL1809)^Channel 14^Input} *)
	STP.XV213A_AlumValveR3_CloseStat AT %IX70.0 : BOOL;	(*  ~ {LinkedWith:TIID^C6920 (EtherCAT)^ScadaRoom_KouplerUTP (EK1100)^ScadaRoom_KouplerFiber (EK1521)^SBR_1 (EK1501)^Term 60 (EL1809)^Channel 15^Input} *)
	STP.XV214A_AlumValveR4_CloseStat AT %IX70.1 : BOOL;	(*  ~ {LinkedWith:TIID^C6920 (EtherCAT)^ScadaRoom_KouplerUTP (EK1100)^ScadaRoom_KouplerFiber (EK1521)^SBR_1 (EK1501)^Term 60 (EL1809)^Channel 16^Input} *)
	STP.XV241A_SludgeValveR1_CloseStat AT %IX70.2 : BOOL;	(*  ~ {LinkedWith:TIID^C6920 (EtherCAT)^ScadaRoom_KouplerUTP (EK1100)^ScadaRoom_KouplerFiber (EK1521)^SBR_1 (EK1501)^Term 61 (EL1809)^Channel 5^Input} *)
	STP.XV242A_SludgeValveR2_CloseStat AT %IX70.3 : BOOL;	(*  ~ {LinkedWith:TIID^C6920 (EtherCAT)^ScadaRoom_KouplerUTP (EK1100)^ScadaRoom_KouplerFiber (EK1521)^SBR_1 (EK1501)^Term 61 (EL1809)^Channel 6^Input} *)
	STP.XV243A_SludgeValveR3_CloseStat AT %IX70.4 : BOOL;	(*  ~ {LinkedWith:TIID^C6920 (EtherCAT)^ScadaRoom_KouplerUTP (EK1100)^ScadaRoom_KouplerFiber (EK1521)^SBR_1 (EK1501)^Term 61 (EL1809)^Channel 7^Input} *)
	STP.XV244A_SludgeValveR4_CloseStat AT %IX70.5 : BOOL;	(*  ~ {LinkedWith:TIID^C6920 (EtherCAT)^ScadaRoom_KouplerUTP (EK1100)^ScadaRoom_KouplerFiber (EK1521)^SBR_1 (EK1501)^Term 61 (EL1809)^Channel 8^Input} *)
	STP.XV241A_SludgeValveR1_OpenStat AT %IX70.6 : BOOL;	(*  ~ {LinkedWith:TIID^C6920 (EtherCAT)^ScadaRoom_KouplerUTP (EK1100)^ScadaRoom_KouplerFiber (EK1521)^SBR_1 (EK1501)^Term 61 (EL1809)^Channel 1^Input} *)
	STP.XV242A_SludgeValveR2_OpenStat AT %IX70.7 : BOOL;	(*  ~ {LinkedWith:TIID^C6920 (EtherCAT)^ScadaRoom_KouplerUTP (EK1100)^ScadaRoom_KouplerFiber (EK1521)^SBR_1 (EK1501)^Term 61 (EL1809)^Channel 2^Input} *)
	STP.XV243A_SludgeValveR3_OpenStat AT %IX71.0 : BOOL;	(*  ~ {LinkedWith:TIID^C6920 (EtherCAT)^ScadaRoom_KouplerUTP (EK1100)^ScadaRoom_KouplerFiber (EK1521)^SBR_1 (EK1501)^Term 61 (EL1809)^Channel 3^Input} *)
	STP.XV244A_SludgeValveR4_OpenStat AT %IX71.1 : BOOL;	(*  ~ {LinkedWith:TIID^C6920 (EtherCAT)^ScadaRoom_KouplerUTP (EK1100)^ScadaRoom_KouplerFiber (EK1521)^SBR_1 (EK1501)^Term 61 (EL1809)^Channel 4^Input} *)
	STP.XV205A_SBRValveR1_OpenCmd AT %QX24.0 : BOOL;	(*  ~ {LinkedWith:TIID^C6920 (EtherCAT)^ScadaRoom_KouplerUTP (EK1100)^ScadaRoom_KouplerFiber (EK1521)^SBR_1 (EK1501)^Term 64 (EL2809)^Channel 1^Output} *)
	STP.XV206A_SBRValveR2_OpenCmd AT %QX24.1 : BOOL;	(*  ~ {LinkedWith:TIID^C6920 (EtherCAT)^ScadaRoom_KouplerUTP (EK1100)^ScadaRoom_KouplerFiber (EK1521)^SBR_1 (EK1501)^Term 64 (EL2809)^Channel 2^Output} *)
	STP.XV207A_SBRValveR3_OpenCmd AT %QX24.2 : BOOL;	(*  ~ {LinkedWith:TIID^C6920 (EtherCAT)^ScadaRoom_KouplerUTP (EK1100)^ScadaRoom_KouplerFiber (EK1521)^SBR_1 (EK1501)^Term 64 (EL2809)^Channel 3^Output} *)
	STP.XV208A_SBRValveR4_OpenCmd AT %QX24.3 : BOOL;	(*  ~ {LinkedWith:TIID^C6920 (EtherCAT)^ScadaRoom_KouplerUTP (EK1100)^ScadaRoom_KouplerFiber (EK1521)^SBR_1 (EK1501)^Term 64 (EL2809)^Channel 4^Output} *)
	STP.XV201A_AirBlowerValveR1_OpenCmd AT %QX24.4 : BOOL;	(*  ~ {LinkedWith:TIID^C6920 (EtherCAT)^ScadaRoom_KouplerUTP (EK1100)^ScadaRoom_KouplerFiber (EK1521)^SBR_1 (EK1501)^Term 64 (EL2809)^Channel 5^Output} *)
	STP.XV202A_AirBlowerValveR2_OpenCmd AT %QX24.5 : BOOL;	(*  ~ {LinkedWith:TIID^C6920 (EtherCAT)^ScadaRoom_KouplerUTP (EK1100)^ScadaRoom_KouplerFiber (EK1521)^SBR_1 (EK1501)^Term 64 (EL2809)^Channel 6^Output} *)
	STP.XV203A_AirBlowerValveR3_OpenCmd AT %QX24.6 : BOOL;	(*  ~ {LinkedWith:TIID^C6920 (EtherCAT)^ScadaRoom_KouplerUTP (EK1100)^ScadaRoom_KouplerFiber (EK1521)^SBR_1 (EK1501)^Term 64 (EL2809)^Channel 7^Output} *)
	STP.XV204A_AirBlowerValveR4_OpenCmd AT %QX24.7 : BOOL;	(*  ~ {LinkedWith:TIID^C6920 (EtherCAT)^ScadaRoom_KouplerUTP (EK1100)^ScadaRoom_KouplerFiber (EK1521)^SBR_1 (EK1501)^Term 64 (EL2809)^Channel 8^Output} *)
	STP.XV221A_LimeValveR1_OpenCmd AT %QX25.0 : BOOL;	(*  ~ {LinkedWith:TIID^C6920 (EtherCAT)^ScadaRoom_KouplerUTP (EK1100)^ScadaRoom_KouplerFiber (EK1521)^SBR_1 (EK1501)^Term 64 (EL2809)^Channel 9^Output} *)
	STP.XV222A_LimeValveR2_OpenCmd AT %QX25.1 : BOOL;	(*  ~ {LinkedWith:TIID^C6920 (EtherCAT)^ScadaRoom_KouplerUTP (EK1100)^ScadaRoom_KouplerFiber (EK1521)^SBR_1 (EK1501)^Term 64 (EL2809)^Channel 10^Output} *)
	STP.XV223A_LimeValveR3_OpenCmd AT %QX25.2 : BOOL;	(*  ~ {LinkedWith:TIID^C6920 (EtherCAT)^ScadaRoom_KouplerUTP (EK1100)^ScadaRoom_KouplerFiber (EK1521)^SBR_1 (EK1501)^Term 64 (EL2809)^Channel 11^Output} *)
	STP.XV224A_LimeValveR4_OpenCmd AT %QX25.3 : BOOL;	(*  ~ {LinkedWith:TIID^C6920 (EtherCAT)^ScadaRoom_KouplerUTP (EK1100)^ScadaRoom_KouplerFiber (EK1521)^SBR_1 (EK1501)^Term 64 (EL2809)^Channel 12^Output} *)
	STP.XV211A_AlumValveR1_OpenCmd AT %QX25.4 : BOOL;	(*  ~ {LinkedWith:TIID^C6920 (EtherCAT)^ScadaRoom_KouplerUTP (EK1100)^ScadaRoom_KouplerFiber (EK1521)^SBR_1 (EK1501)^Term 64 (EL2809)^Channel 13^Output} *)
	STP.XV212A_AlumValveR2_OpenCmd AT %QX25.5 : BOOL;	(*  ~ {LinkedWith:TIID^C6920 (EtherCAT)^ScadaRoom_KouplerUTP (EK1100)^ScadaRoom_KouplerFiber (EK1521)^SBR_1 (EK1501)^Term 64 (EL2809)^Channel 14^Output} *)
	STP.XV213A_AlumValveR3_OpenCmd AT %QX25.6 : BOOL;	(*  ~ {LinkedWith:TIID^C6920 (EtherCAT)^ScadaRoom_KouplerUTP (EK1100)^ScadaRoom_KouplerFiber (EK1521)^SBR_1 (EK1501)^Term 64 (EL2809)^Channel 15^Output} *)
	STP.XV214A_AlumValveR4_OpenCmd AT %QX25.7 : BOOL;	(*  ~ {LinkedWith:TIID^C6920 (EtherCAT)^ScadaRoom_KouplerUTP (EK1100)^ScadaRoom_KouplerFiber (EK1521)^SBR_1 (EK1501)^Term 64 (EL2809)^Channel 16^Output} *)
	STP.XV241A_SludgeValveR1_OpenCmd AT %QX26.0 : BOOL;	(*  ~ {LinkedWith:TIID^C6920 (EtherCAT)^ScadaRoom_KouplerUTP (EK1100)^ScadaRoom_KouplerFiber (EK1521)^SBR_1 (EK1501)^Term 65 (EL2809)^Channel 1^Output} *)
	STP.XV242A_SludgeValveR2_OpenCmd AT %QX26.1 : BOOL;	(*  ~ {LinkedWith:TIID^C6920 (EtherCAT)^ScadaRoom_KouplerUTP (EK1100)^ScadaRoom_KouplerFiber (EK1521)^SBR_1 (EK1501)^Term 65 (EL2809)^Channel 2^Output} *)
	STP.XV243A_SludgeValveR3_OpenCmd AT %QX26.2 : BOOL;	(*  ~ {LinkedWith:TIID^C6920 (EtherCAT)^ScadaRoom_KouplerUTP (EK1100)^ScadaRoom_KouplerFiber (EK1521)^SBR_1 (EK1501)^Term 65 (EL2809)^Channel 3^Output} *)
	STP.XV244A_SludgeValveR4_OpenCmd AT %QX26.3 : BOOL;	(*  ~ {LinkedWith:TIID^C6920 (EtherCAT)^ScadaRoom_KouplerUTP (EK1100)^ScadaRoom_KouplerFiber (EK1521)^SBR_1 (EK1501)^Term 65 (EL2809)^Channel 4^Output} *)
	STP.XV241A_SludgeValveR1_CloseCmd AT %QX26.4 : BOOL;	(*  ~ {LinkedWith:TIID^C6920 (EtherCAT)^ScadaRoom_KouplerUTP (EK1100)^ScadaRoom_KouplerFiber (EK1521)^SBR_1 (EK1501)^Term 65 (EL2809)^Channel 5^Output} *)
	STP.XV242A_SludgeValveR2_CloseCmd AT %QX26.5 : BOOL;	(*  ~ {LinkedWith:TIID^C6920 (EtherCAT)^ScadaRoom_KouplerUTP (EK1100)^ScadaRoom_KouplerFiber (EK1521)^SBR_1 (EK1501)^Term 65 (EL2809)^Channel 6^Output} *)
	STP.XV243A_SludgeValveR3_CloseCmd AT %QX26.6 : BOOL;	(*  ~ {LinkedWith:TIID^C6920 (EtherCAT)^ScadaRoom_KouplerUTP (EK1100)^ScadaRoom_KouplerFiber (EK1521)^SBR_1 (EK1501)^Term 65 (EL2809)^Channel 7^Output} *)
	STP.XV244A_SludgeValveR4_CloseCmd AT %QX26.7 : BOOL;	(*  ~ {LinkedWith:TIID^C6920 (EtherCAT)^ScadaRoom_KouplerUTP (EK1100)^ScadaRoom_KouplerFiber (EK1521)^SBR_1 (EK1501)^Term 65 (EL2809)^Channel 8^Output} *)
	STP.XV205A_SBRValveR1_CloseCmd AT %QX27.0 : BOOL;	(*  ~ {LinkedWith:TIID^C6920 (EtherCAT)^ScadaRoom_KouplerUTP (EK1100)^ScadaRoom_KouplerFiber (EK1521)^SBR_1 (EK1501)^Term 66 (EL2809)^Channel 1^Output} *)
	STP.XV206A_SBRValveR2_CloseCmd AT %QX27.1 : BOOL;	(*  ~ {LinkedWith:TIID^C6920 (EtherCAT)^ScadaRoom_KouplerUTP (EK1100)^ScadaRoom_KouplerFiber (EK1521)^SBR_1 (EK1501)^Term 66 (EL2809)^Channel 2^Output} *)
	STP.XV207A_SBRValveR3_CloseCmd AT %QX27.2 : BOOL;	(*  ~ {LinkedWith:TIID^C6920 (EtherCAT)^ScadaRoom_KouplerUTP (EK1100)^ScadaRoom_KouplerFiber (EK1521)^SBR_1 (EK1501)^Term 66 (EL2809)^Channel 3^Output} *)
	STP.XV208A_SBRValveR4_CloseCmd AT %QX27.3 : BOOL;	(*  ~ {LinkedWith:TIID^C6920 (EtherCAT)^ScadaRoom_KouplerUTP (EK1100)^ScadaRoom_KouplerFiber (EK1521)^SBR_1 (EK1501)^Term 66 (EL2809)^Channel 4^Output} *)
	STP.XV201A_AirBlowerValveR1_CloseCmd AT %QX27.4 : BOOL;	(*  ~ {LinkedWith:TIID^C6920 (EtherCAT)^ScadaRoom_KouplerUTP (EK1100)^ScadaRoom_KouplerFiber (EK1521)^SBR_1 (EK1501)^Term 66 (EL2809)^Channel 5^Output} *)
	STP.XV202A_AirBlowerValveR2_CloseCmd AT %QX27.5 : BOOL;	(*  ~ {LinkedWith:TIID^C6920 (EtherCAT)^ScadaRoom_KouplerUTP (EK1100)^ScadaRoom_KouplerFiber (EK1521)^SBR_1 (EK1501)^Term 66 (EL2809)^Channel 6^Output} *)
	STP.XV203A_AirBlowerValveR3_CloseCmd AT %QX27.6 : BOOL;	(*  ~ {LinkedWith:TIID^C6920 (EtherCAT)^ScadaRoom_KouplerUTP (EK1100)^ScadaRoom_KouplerFiber (EK1521)^SBR_1 (EK1501)^Term 66 (EL2809)^Channel 7^Output} *)
	STP.XV204A_AirBlowerValveR4_CloseCmd AT %QX27.7 : BOOL;	(*  ~ {LinkedWith:TIID^C6920 (EtherCAT)^ScadaRoom_KouplerUTP (EK1100)^ScadaRoom_KouplerFiber (EK1521)^SBR_1 (EK1501)^Term 66 (EL2809)^Channel 8^Output} *)
	STP.XV221A_LimeValveR1_CloseCmd AT %QX28.0 : BOOL;	(*  ~ {LinkedWith:TIID^C6920 (EtherCAT)^ScadaRoom_KouplerUTP (EK1100)^ScadaRoom_KouplerFiber (EK1521)^SBR_1 (EK1501)^Term 66 (EL2809)^Channel 9^Output} *)
	STP.XV222A_LimeValveR2_CloseCmd AT %QX28.1 : BOOL;	(*  ~ {LinkedWith:TIID^C6920 (EtherCAT)^ScadaRoom_KouplerUTP (EK1100)^ScadaRoom_KouplerFiber (EK1521)^SBR_1 (EK1501)^Term 66 (EL2809)^Channel 10^Output} *)
	STP.XV223A_LimeValveR3_CloseCmd AT %QX28.2 : BOOL;	(*  ~ {LinkedWith:TIID^C6920 (EtherCAT)^ScadaRoom_KouplerUTP (EK1100)^ScadaRoom_KouplerFiber (EK1521)^SBR_1 (EK1501)^Term 66 (EL2809)^Channel 11^Output} *)
	STP.XV224A_LimeValveR4_CloseCmd AT %QX28.3 : BOOL;	(*  ~ {LinkedWith:TIID^C6920 (EtherCAT)^ScadaRoom_KouplerUTP (EK1100)^ScadaRoom_KouplerFiber (EK1521)^SBR_1 (EK1501)^Term 66 (EL2809)^Channel 12^Output} *)
	STP.XV211A_AlumValveR1_CloseCmd AT %QX28.4 : BOOL;	(*  ~ {LinkedWith:TIID^C6920 (EtherCAT)^ScadaRoom_KouplerUTP (EK1100)^ScadaRoom_KouplerFiber (EK1521)^SBR_1 (EK1501)^Term 66 (EL2809)^Channel 13^Output} *)
	STP.XV212A_AlumValveR2_CloseCmd AT %QX28.5 : BOOL;	(*  ~ {LinkedWith:TIID^C6920 (EtherCAT)^ScadaRoom_KouplerUTP (EK1100)^ScadaRoom_KouplerFiber (EK1521)^SBR_1 (EK1501)^Term 66 (EL2809)^Channel 14^Output} *)
	STP.XV213A_AlumValveR3_CloseCmd AT %QX28.6 : BOOL;	(*  ~ {LinkedWith:TIID^C6920 (EtherCAT)^ScadaRoom_KouplerUTP (EK1100)^ScadaRoom_KouplerFiber (EK1521)^SBR_1 (EK1501)^Term 66 (EL2809)^Channel 15^Output} *)
	STP.XV214A_AlumValveR4_CloseCmd AT %QX28.7 : BOOL;	(*  ~ {LinkedWith:TIID^C6920 (EtherCAT)^ScadaRoom_KouplerUTP (EK1100)^ScadaRoom_KouplerFiber (EK1521)^SBR_1 (EK1501)^Term 66 (EL2809)^Channel 16^Output} *)
	STP.OPR1AON_ReactorR1_OnlineCmd AT %QX29.0 : BOOL;	(*  ~ {LinkedWith:TIID^C6920 (EtherCAT)^ScadaRoom_KouplerUTP (EK1100)^ScadaRoom_KouplerFiber (EK1521)^SBR_1 (EK1501)^Term 67 (EL2809)^Channel 1^Output} *)
	STP.OPR2AON_ReactorR2_OnlineCmd AT %QX29.1 : BOOL;	(*  ~ {LinkedWith:TIID^C6920 (EtherCAT)^ScadaRoom_KouplerUTP (EK1100)^ScadaRoom_KouplerFiber (EK1521)^SBR_1 (EK1501)^Term 67 (EL2809)^Channel 2^Output} *)
	STP.OPR3AON_ReactorR3_OnlineCmd AT %QX29.2 : BOOL;	(*  ~ {LinkedWith:TIID^C6920 (EtherCAT)^ScadaRoom_KouplerUTP (EK1100)^ScadaRoom_KouplerFiber (EK1521)^SBR_1 (EK1501)^Term 67 (EL2809)^Channel 3^Output} *)
	STP.OPR4AON_ReactorR4_OnlineCmd AT %QX29.3 : BOOL;	(*  ~ {LinkedWith:TIID^C6920 (EtherCAT)^ScadaRoom_KouplerUTP (EK1100)^ScadaRoom_KouplerFiber (EK1521)^SBR_1 (EK1501)^Term 67 (EL2809)^Channel 4^Output} *)
	STP.OPR1AOFF_ReactorR1_OfflineCmd AT %QX29.4 : BOOL;	(*  ~ {LinkedWith:TIID^C6920 (EtherCAT)^ScadaRoom_KouplerUTP (EK1100)^ScadaRoom_KouplerFiber (EK1521)^SBR_1 (EK1501)^Term 67 (EL2809)^Channel 5^Output} *)
	STP.OPR2AOFF_ReactorR2_OfflineCmd AT %QX29.5 : BOOL;	(*  ~ {LinkedWith:TIID^C6920 (EtherCAT)^ScadaRoom_KouplerUTP (EK1100)^ScadaRoom_KouplerFiber (EK1521)^SBR_1 (EK1501)^Term 67 (EL2809)^Channel 6^Output} *)
	STP.OPR3AOFF_ReactorR3_OfflineCmd AT %QX29.6 : BOOL;	(*  ~ {LinkedWith:TIID^C6920 (EtherCAT)^ScadaRoom_KouplerUTP (EK1100)^ScadaRoom_KouplerFiber (EK1521)^SBR_1 (EK1501)^Term 67 (EL2809)^Channel 7^Output} *)
	STP.OPR4AOFF_ReactorR4_OfflineCmd AT %QX29.7 : BOOL;	(*  ~ {LinkedWith:TIID^C6920 (EtherCAT)^ScadaRoom_KouplerUTP (EK1100)^ScadaRoom_KouplerFiber (EK1521)^SBR_1 (EK1501)^Term 67 (EL2809)^Channel 8^Output} *)
	STP.OPR1ASW_ReactorR1_SwitchCmd AT %QX30.0 : BOOL;	(*  ~ {LinkedWith:TIID^C6920 (EtherCAT)^ScadaRoom_KouplerUTP (EK1100)^ScadaRoom_KouplerFiber (EK1521)^SBR_1 (EK1501)^Term 68 (EL2809)^Channel 1^Output} *)
	STP.OPR2ASW_ReactorR2_SwitchCmd AT %QX30.1 : BOOL;	(*  ~ {LinkedWith:TIID^C6920 (EtherCAT)^ScadaRoom_KouplerUTP (EK1100)^ScadaRoom_KouplerFiber (EK1521)^SBR_1 (EK1501)^Term 68 (EL2809)^Channel 2^Output} *)
	STP.OPR3ASW_ReactorR3_SwitchCmd AT %QX30.2 : BOOL;	(*  ~ {LinkedWith:TIID^C6920 (EtherCAT)^ScadaRoom_KouplerUTP (EK1100)^ScadaRoom_KouplerFiber (EK1521)^SBR_1 (EK1501)^Term 68 (EL2809)^Channel 3^Output} *)
	STP.OPR4ASW_ReactorR4_SwitchCmd AT %QX30.3 : BOOL;	(*  ~ {LinkedWith:TIID^C6920 (EtherCAT)^ScadaRoom_KouplerUTP (EK1100)^ScadaRoom_KouplerFiber (EK1521)^SBR_1 (EK1501)^Term 68 (EL2809)^Channel 4^Output} *)
	STP.AUX402_PLCRunStat AT %QX72.5 : BOOL;	(*  ~ {LinkedWith:TIID^C6920 (EtherCAT)^ScadaRoom_KouplerUTP (EK1100)^ScadaRoom_KouplerFiber (EK1521)^SBR_1 (EK1501)^Term 68 (EL2809)^Channel 5^Output} *)
	STP.AUX401_CommonAlarm AT %QX72.6 : BOOL;	(*  ~ {LinkedWith:TIID^C6920 (EtherCAT)^ScadaRoom_KouplerUTP (EK1100)^ScadaRoom_KouplerFiber (EK1521)^SBR_1 (EK1501)^Term 68 (EL2809)^Channel 6^Output} *)
	STP.LSH201B1_LevelSensorR1 AT %IX72.2 : BOOL;	(*  ~ {LinkedWith:TIID^C6920 (EtherCAT)^ScadaRoom_KouplerUTP (EK1100)^ScadaRoom_KouplerFiber (EK1521)^SBR_2 (EK1501)^Term 70 (EL1809)^Channel 1^Input} *)
	STP.LSH201B2_LevelSensorR2 AT %IX72.3 : BOOL;	(*  ~ {LinkedWith:TIID^C6920 (EtherCAT)^ScadaRoom_KouplerUTP (EK1100)^ScadaRoom_KouplerFiber (EK1521)^SBR_2 (EK1501)^Term 70 (EL1809)^Channel 2^Input} *)
	STP.LSH201B3_LevelSensorR3 AT %IX72.4 : BOOL;	(*  ~ {LinkedWith:TIID^C6920 (EtherCAT)^ScadaRoom_KouplerUTP (EK1100)^ScadaRoom_KouplerFiber (EK1521)^SBR_2 (EK1501)^Term 70 (EL1809)^Channel 3^Input} *)
	STP.LSH201B4_LevelSensorR4 AT %IX72.5 : BOOL;	(*  ~ {LinkedWith:TIID^C6920 (EtherCAT)^ScadaRoom_KouplerUTP (EK1100)^ScadaRoom_KouplerFiber (EK1521)^SBR_2 (EK1501)^Term 70 (EL1809)^Channel 4^Input} *)
	STP.OPR1B_ReactorStatus AT %IX72.6 : BOOL;	(*  ~ {LinkedWith:TIID^C6920 (EtherCAT)^ScadaRoom_KouplerUTP (EK1100)^ScadaRoom_KouplerFiber (EK1521)^SBR_2 (EK1501)^Term 70 (EL1809)^Channel 5^Input} *)
	STP.OPR2B_ReactorStatus AT %IX72.7 : BOOL;	(*  ~ {LinkedWith:TIID^C6920 (EtherCAT)^ScadaRoom_KouplerUTP (EK1100)^ScadaRoom_KouplerFiber (EK1521)^SBR_2 (EK1501)^Term 70 (EL1809)^Channel 6^Input} *)
	STP.OPR3B_ReactorStatus AT %IX73.0 : BOOL;	(*  ~ {LinkedWith:TIID^C6920 (EtherCAT)^ScadaRoom_KouplerUTP (EK1100)^ScadaRoom_KouplerFiber (EK1521)^SBR_2 (EK1501)^Term 70 (EL1809)^Channel 7^Input} *)
	STP.OPR4B_ReactorStatus AT %IX73.1 : BOOL;	(*  ~ {LinkedWith:TIID^C6920 (EtherCAT)^ScadaRoom_KouplerUTP (EK1100)^ScadaRoom_KouplerFiber (EK1521)^SBR_2 (EK1501)^Term 70 (EL1809)^Channel 8^Input} *)
	STP.DP05_DoorPanelStatus AT %IX73.2 : BOOL;	(*  ~ {LinkedWith:TIID^C6920 (EtherCAT)^ScadaRoom_KouplerUTP (EK1100)^ScadaRoom_KouplerFiber (EK1521)^SBR_2 (EK1501)^Term 70 (EL1809)^Channel 9^Input} *)
	STP.TMT05_FanStatus AT %IX73.3 : BOOL;	(*  ~ {LinkedWith:TIID^C6920 (EtherCAT)^ScadaRoom_KouplerUTP (EK1100)^ScadaRoom_KouplerFiber (EK1521)^SBR_2 (EK1501)^Term 70 (EL1809)^Channel 10^Input} *)
	STP.HR201B1_DecantHighLevelR1 AT %IX73.4 : BOOL;	(*  ~ {LinkedWith:TIID^C6920 (EtherCAT)^ScadaRoom_KouplerUTP (EK1100)^ScadaRoom_KouplerFiber (EK1521)^SBR_2 (EK1501)^Term 71 (EL1809)^Channel 1^Input} *)
	STP.LR201B1_DecantLowLevelR1 AT %IX73.5 : BOOL;	(*  ~ {LinkedWith:TIID^C6920 (EtherCAT)^ScadaRoom_KouplerUTP (EK1100)^ScadaRoom_KouplerFiber (EK1521)^SBR_2 (EK1501)^Term 71 (EL1809)^Channel 2^Input} *)
	STP.HR201B2_DecantHighLevelR2 AT %IX73.6 : BOOL;	(*  ~ {LinkedWith:TIID^C6920 (EtherCAT)^ScadaRoom_KouplerUTP (EK1100)^ScadaRoom_KouplerFiber (EK1521)^SBR_2 (EK1501)^Term 71 (EL1809)^Channel 3^Input} *)
	STP.LR201B2_DecantLowLevelR2 AT %IX73.7 : BOOL;	(*  ~ {LinkedWith:TIID^C6920 (EtherCAT)^ScadaRoom_KouplerUTP (EK1100)^ScadaRoom_KouplerFiber (EK1521)^SBR_2 (EK1501)^Term 71 (EL1809)^Channel 4^Input} *)
	STP.HR201B3_DecantHighLevelR3 AT %IX74.0 : BOOL;	(*  ~ {LinkedWith:TIID^C6920 (EtherCAT)^ScadaRoom_KouplerUTP (EK1100)^ScadaRoom_KouplerFiber (EK1521)^SBR_2 (EK1501)^Term 71 (EL1809)^Channel 5^Input} *)
	STP.HR201B4_DecantHighLevelR4 AT %IX74.1 : BOOL;	(*  ~ {LinkedWith:TIID^C6920 (EtherCAT)^ScadaRoom_KouplerUTP (EK1100)^ScadaRoom_KouplerFiber (EK1521)^SBR_2 (EK1501)^Term 71 (EL1809)^Channel 7^Input} *)
	STP.LR201B3_DecantLowLevelR3 AT %IX74.2 : BOOL;	(*  ~ {LinkedWith:TIID^C6920 (EtherCAT)^ScadaRoom_KouplerUTP (EK1100)^ScadaRoom_KouplerFiber (EK1521)^SBR_2 (EK1501)^Term 71 (EL1809)^Channel 6^Input} *)
	STP.LR201B4_DecantLowLevelR4 AT %IX74.3 : BOOL;	(*  ~ {LinkedWith:TIID^C6920 (EtherCAT)^ScadaRoom_KouplerUTP (EK1100)^ScadaRoom_KouplerFiber (EK1521)^SBR_2 (EK1501)^Term 71 (EL1809)^Channel 8^Input} *)
	STP.XV205B_SBRValveR1_OpenStat AT %IX74.4 : BOOL;	(*  ~ {LinkedWith:TIID^C6920 (EtherCAT)^ScadaRoom_KouplerUTP (EK1100)^ScadaRoom_KouplerFiber (EK1521)^SBR_2 (EK1501)^Term 72 (EL1809)^Channel 1^Input} *)
	STP.XV206B_SBRValveR2_OpenStat AT %IX74.5 : BOOL;	(*  ~ {LinkedWith:TIID^C6920 (EtherCAT)^ScadaRoom_KouplerUTP (EK1100)^ScadaRoom_KouplerFiber (EK1521)^SBR_2 (EK1501)^Term 72 (EL1809)^Channel 2^Input} *)
	STP.XV207B_SBRValveR3_OpenStat AT %IX74.6 : BOOL;	(*  ~ {LinkedWith:TIID^C6920 (EtherCAT)^ScadaRoom_KouplerUTP (EK1100)^ScadaRoom_KouplerFiber (EK1521)^SBR_2 (EK1501)^Term 72 (EL1809)^Channel 3^Input} *)
	STP.XV208B_SBRValveR4_OpenStat AT %IX74.7 : BOOL;	(*  ~ {LinkedWith:TIID^C6920 (EtherCAT)^ScadaRoom_KouplerUTP (EK1100)^ScadaRoom_KouplerFiber (EK1521)^SBR_2 (EK1501)^Term 72 (EL1809)^Channel 4^Input} *)
	STP.XV201B_AirBlowerValveR1_OpenStat AT %IX75.0 : BOOL;	(*  ~ {LinkedWith:TIID^C6920 (EtherCAT)^ScadaRoom_KouplerUTP (EK1100)^ScadaRoom_KouplerFiber (EK1521)^SBR_2 (EK1501)^Term 72 (EL1809)^Channel 5^Input} *)
	STP.XV202B_AirBlowerValveR2_OpenStat AT %IX75.1 : BOOL;	(*  ~ {LinkedWith:TIID^C6920 (EtherCAT)^ScadaRoom_KouplerUTP (EK1100)^ScadaRoom_KouplerFiber (EK1521)^SBR_2 (EK1501)^Term 72 (EL1809)^Channel 6^Input} *)
	STP.XV203B_AirBlowerValveR3_OpenStat AT %IX75.2 : BOOL;	(*  ~ {LinkedWith:TIID^C6920 (EtherCAT)^ScadaRoom_KouplerUTP (EK1100)^ScadaRoom_KouplerFiber (EK1521)^SBR_2 (EK1501)^Term 72 (EL1809)^Channel 7^Input} *)
	STP.XV204B_AirBlowerValveR4_OpenStat AT %IX75.3 : BOOL;	(*  ~ {LinkedWith:TIID^C6920 (EtherCAT)^ScadaRoom_KouplerUTP (EK1100)^ScadaRoom_KouplerFiber (EK1521)^SBR_2 (EK1501)^Term 72 (EL1809)^Channel 8^Input} *)
	STP.XV221B_LimeValveR1_OpenStat AT %IX75.4 : BOOL;	(*  ~ {LinkedWith:TIID^C6920 (EtherCAT)^ScadaRoom_KouplerUTP (EK1100)^ScadaRoom_KouplerFiber (EK1521)^SBR_2 (EK1501)^Term 72 (EL1809)^Channel 9^Input} *)
	STP.XV222B_LimeValveR2_OpenStat AT %IX75.5 : BOOL;	(*  ~ {LinkedWith:TIID^C6920 (EtherCAT)^ScadaRoom_KouplerUTP (EK1100)^ScadaRoom_KouplerFiber (EK1521)^SBR_2 (EK1501)^Term 72 (EL1809)^Channel 10^Input} *)
	STP.XV223B_LimeValveR3_OpenStat AT %IX75.6 : BOOL;	(*  ~ {LinkedWith:TIID^C6920 (EtherCAT)^ScadaRoom_KouplerUTP (EK1100)^ScadaRoom_KouplerFiber (EK1521)^SBR_2 (EK1501)^Term 72 (EL1809)^Channel 11^Input} *)
	STP.XV224B_LimeValveR4_OpenStat AT %IX75.7 : BOOL;	(*  ~ {LinkedWith:TIID^C6920 (EtherCAT)^ScadaRoom_KouplerUTP (EK1100)^ScadaRoom_KouplerFiber (EK1521)^SBR_2 (EK1501)^Term 72 (EL1809)^Channel 12^Input} *)
	STP.XV211B_AlumValveR1_OpenStat AT %IX76.0 : BOOL;	(*  ~ {LinkedWith:TIID^C6920 (EtherCAT)^ScadaRoom_KouplerUTP (EK1100)^ScadaRoom_KouplerFiber (EK1521)^SBR_2 (EK1501)^Term 72 (EL1809)^Channel 13^Input} *)
	STP.XV212B_AlumValveR2_OpenStat AT %IX76.1 : BOOL;	(*  ~ {LinkedWith:TIID^C6920 (EtherCAT)^ScadaRoom_KouplerUTP (EK1100)^ScadaRoom_KouplerFiber (EK1521)^SBR_2 (EK1501)^Term 72 (EL1809)^Channel 14^Input} *)
	STP.XV213B_AlumValveR3_OpenStat AT %IX76.2 : BOOL;	(*  ~ {LinkedWith:TIID^C6920 (EtherCAT)^ScadaRoom_KouplerUTP (EK1100)^ScadaRoom_KouplerFiber (EK1521)^SBR_2 (EK1501)^Term 72 (EL1809)^Channel 15^Input} *)
	STP.XV214B_AlumValveR4_OpenStat AT %IX76.3 : BOOL;	(*  ~ {LinkedWith:TIID^C6920 (EtherCAT)^ScadaRoom_KouplerUTP (EK1100)^ScadaRoom_KouplerFiber (EK1521)^SBR_2 (EK1501)^Term 72 (EL1809)^Channel 16^Input} *)
	STP.XV205B_SBRValveR1_CloseStat AT %IX76.4 : BOOL;	(*  ~ {LinkedWith:TIID^C6920 (EtherCAT)^ScadaRoom_KouplerUTP (EK1100)^ScadaRoom_KouplerFiber (EK1521)^SBR_2 (EK1501)^Term 73 (EL1809)^Channel 1^Input} *)
	STP.XV206B_SBRValveR2_CloseStat AT %IX76.5 : BOOL;	(*  ~ {LinkedWith:TIID^C6920 (EtherCAT)^ScadaRoom_KouplerUTP (EK1100)^ScadaRoom_KouplerFiber (EK1521)^SBR_2 (EK1501)^Term 73 (EL1809)^Channel 2^Input} *)
	STP.XV207B_SBRValveR3_CloseStat AT %IX76.6 : BOOL;	(*  ~ {LinkedWith:TIID^C6920 (EtherCAT)^ScadaRoom_KouplerUTP (EK1100)^ScadaRoom_KouplerFiber (EK1521)^SBR_2 (EK1501)^Term 73 (EL1809)^Channel 3^Input} *)
	STP.XV208B_SBRValveR4_CloseStat AT %IX76.7 : BOOL;	(*  ~ {LinkedWith:TIID^C6920 (EtherCAT)^ScadaRoom_KouplerUTP (EK1100)^ScadaRoom_KouplerFiber (EK1521)^SBR_2 (EK1501)^Term 73 (EL1809)^Channel 4^Input} *)
	STP.XV201B_AirBlowerValveR1_CloseStat AT %IX77.0 : BOOL;	(*  ~ {LinkedWith:TIID^C6920 (EtherCAT)^ScadaRoom_KouplerUTP (EK1100)^ScadaRoom_KouplerFiber (EK1521)^SBR_2 (EK1501)^Term 73 (EL1809)^Channel 5^Input} *)
	STP.XV202B_AirBlowerValveR2_CloseStat AT %IX77.1 : BOOL;	(*  ~ {LinkedWith:TIID^C6920 (EtherCAT)^ScadaRoom_KouplerUTP (EK1100)^ScadaRoom_KouplerFiber (EK1521)^SBR_2 (EK1501)^Term 73 (EL1809)^Channel 6^Input} *)
	STP.XV203B_AirBlowerValveR3_CloseStat AT %IX77.2 : BOOL;	(*  ~ {LinkedWith:TIID^C6920 (EtherCAT)^ScadaRoom_KouplerUTP (EK1100)^ScadaRoom_KouplerFiber (EK1521)^SBR_2 (EK1501)^Term 73 (EL1809)^Channel 7^Input} *)
	STP.XV204B_AirBlowerValveR4_CloseStat AT %IX77.3 : BOOL;	(*  ~ {LinkedWith:TIID^C6920 (EtherCAT)^ScadaRoom_KouplerUTP (EK1100)^ScadaRoom_KouplerFiber (EK1521)^SBR_2 (EK1501)^Term 73 (EL1809)^Channel 8^Input} *)
	STP.XV221B_LimeValveR1_CloseStat AT %IX77.4 : BOOL;	(*  ~ {LinkedWith:TIID^C6920 (EtherCAT)^ScadaRoom_KouplerUTP (EK1100)^ScadaRoom_KouplerFiber (EK1521)^SBR_2 (EK1501)^Term 73 (EL1809)^Channel 9^Input} *)
	STP.XV222B_LimeValveR2_CloseStat AT %IX77.5 : BOOL;	(*  ~ {LinkedWith:TIID^C6920 (EtherCAT)^ScadaRoom_KouplerUTP (EK1100)^ScadaRoom_KouplerFiber (EK1521)^SBR_2 (EK1501)^Term 73 (EL1809)^Channel 10^Input} *)
	STP.XV223B_LimeValveR3_CloseStat AT %IX77.6 : BOOL;	(*  ~ {LinkedWith:TIID^C6920 (EtherCAT)^ScadaRoom_KouplerUTP (EK1100)^ScadaRoom_KouplerFiber (EK1521)^SBR_2 (EK1501)^Term 73 (EL1809)^Channel 11^Input} *)
	STP.XV224B_LimeValveR4_CloseStat AT %IX77.7 : BOOL;	(*  ~ {LinkedWith:TIID^C6920 (EtherCAT)^ScadaRoom_KouplerUTP (EK1100)^ScadaRoom_KouplerFiber (EK1521)^SBR_2 (EK1501)^Term 73 (EL1809)^Channel 12^Input} *)
	STP.XV211B_AlumValveR1_CloseStat AT %IX78.0 : BOOL;	(*  ~ {LinkedWith:TIID^C6920 (EtherCAT)^ScadaRoom_KouplerUTP (EK1100)^ScadaRoom_KouplerFiber (EK1521)^SBR_2 (EK1501)^Term 73 (EL1809)^Channel 13^Input} *)
	STP.XV212B_AlumValveR2_CloseStat AT %IX78.1 : BOOL;	(*  ~ {LinkedWith:TIID^C6920 (EtherCAT)^ScadaRoom_KouplerUTP (EK1100)^ScadaRoom_KouplerFiber (EK1521)^SBR_2 (EK1501)^Term 73 (EL1809)^Channel 14^Input} *)
	STP.XV213B_AlumValveR3_CloseStat AT %IX78.2 : BOOL;	(*  ~ {LinkedWith:TIID^C6920 (EtherCAT)^ScadaRoom_KouplerUTP (EK1100)^ScadaRoom_KouplerFiber (EK1521)^SBR_2 (EK1501)^Term 73 (EL1809)^Channel 15^Input} *)
	STP.XV214B_AlumValveR4_CloseStat AT %IX78.3 : BOOL;	(*  ~ {LinkedWith:TIID^C6920 (EtherCAT)^ScadaRoom_KouplerUTP (EK1100)^ScadaRoom_KouplerFiber (EK1521)^SBR_2 (EK1501)^Term 73 (EL1809)^Channel 16^Input} *)
	STP.XV20xB_SludgeValveR1_CloseStat AT %IX78.4 : BOOL;	(*  ~ {LinkedWith:TIID^C6920 (EtherCAT)^ScadaRoom_KouplerUTP (EK1100)^ScadaRoom_KouplerFiber (EK1521)^SBR_2 (EK1501)^Term 74 (EL1809)^Channel 1^Input} *)
	STP.XV20xB_SludgeValveR2_CloseStat AT %IX78.5 : BOOL;	(*  ~ {LinkedWith:TIID^C6920 (EtherCAT)^ScadaRoom_KouplerUTP (EK1100)^ScadaRoom_KouplerFiber (EK1521)^SBR_2 (EK1501)^Term 74 (EL1809)^Channel 2^Input} *)
	STP.XV20xB_SludgeValveR3_CloseStat AT %IX78.6 : BOOL;	(*  ~ {LinkedWith:TIID^C6920 (EtherCAT)^ScadaRoom_KouplerUTP (EK1100)^ScadaRoom_KouplerFiber (EK1521)^SBR_2 (EK1501)^Term 74 (EL1809)^Channel 3^Input} *)
	STP.XV20xB_SludgeValveR4_CloseStat AT %IX78.7 : BOOL;	(*  ~ {LinkedWith:TIID^C6920 (EtherCAT)^ScadaRoom_KouplerUTP (EK1100)^ScadaRoom_KouplerFiber (EK1521)^SBR_2 (EK1501)^Term 74 (EL1809)^Channel 4^Input} *)
	STP.XV20xB_SludgeValveR1_OpenStat AT %IX79.0 : BOOL;	(*  ~ {LinkedWith:TIID^C6920 (EtherCAT)^ScadaRoom_KouplerUTP (EK1100)^ScadaRoom_KouplerFiber (EK1521)^SBR_2 (EK1501)^Term 74 (EL1809)^Channel 5^Input} *)
	STP.XV20xB_SludgeValveR2_OpenStat AT %IX79.1 : BOOL;	(*  ~ {LinkedWith:TIID^C6920 (EtherCAT)^ScadaRoom_KouplerUTP (EK1100)^ScadaRoom_KouplerFiber (EK1521)^SBR_2 (EK1501)^Term 74 (EL1809)^Channel 6^Input} *)
	STP.XV20xB_SludgeValveR3_OpenStat AT %IX79.2 : BOOL;	(*  ~ {LinkedWith:TIID^C6920 (EtherCAT)^ScadaRoom_KouplerUTP (EK1100)^ScadaRoom_KouplerFiber (EK1521)^SBR_2 (EK1501)^Term 74 (EL1809)^Channel 7^Input} *)
	STP.XV20xB_SludgeValveR4_OpenStat AT %IX79.3 : BOOL;	(*  ~ {LinkedWith:TIID^C6920 (EtherCAT)^ScadaRoom_KouplerUTP (EK1100)^ScadaRoom_KouplerFiber (EK1521)^SBR_2 (EK1501)^Term 74 (EL1809)^Channel 8^Input} *)
	STP.XV205B_SBRValveR1_OpenCmd AT %QX30.6 : BOOL;	(*  ~ {LinkedWith:TIID^C6920 (EtherCAT)^ScadaRoom_KouplerUTP (EK1100)^ScadaRoom_KouplerFiber (EK1521)^SBR_2 (EK1501)^Term 77 (EL2809)^Channel 1^Output} *)
	STP.XV206B_SBRValveR2_OpenCmd AT %QX30.7 : BOOL;	(*  ~ {LinkedWith:TIID^C6920 (EtherCAT)^ScadaRoom_KouplerUTP (EK1100)^ScadaRoom_KouplerFiber (EK1521)^SBR_2 (EK1501)^Term 77 (EL2809)^Channel 2^Output} *)
	STP.XV207B_SBRValveR3_OpenCmd AT %QX31.0 : BOOL;	(*  ~ {LinkedWith:TIID^C6920 (EtherCAT)^ScadaRoom_KouplerUTP (EK1100)^ScadaRoom_KouplerFiber (EK1521)^SBR_2 (EK1501)^Term 77 (EL2809)^Channel 3^Output} *)
	STP.XV208B_SBRValveR4_OpenCmd AT %QX31.1 : BOOL;	(*  ~ {LinkedWith:TIID^C6920 (EtherCAT)^ScadaRoom_KouplerUTP (EK1100)^ScadaRoom_KouplerFiber (EK1521)^SBR_2 (EK1501)^Term 77 (EL2809)^Channel 4^Output} *)
	STP.XV202B_AirBlowerValveR2_OpenCmd AT %QX31.3 : BOOL;	(*  ~ {LinkedWith:TIID^C6920 (EtherCAT)^ScadaRoom_KouplerUTP (EK1100)^ScadaRoom_KouplerFiber (EK1521)^SBR_2 (EK1501)^Term 77 (EL2809)^Channel 6^Output} *)
	STP.XV201B_AirBlowerValveR1_OpenCmd AT %QX31.2 : BOOL;	(*  ~ {LinkedWith:TIID^C6920 (EtherCAT)^ScadaRoom_KouplerUTP (EK1100)^ScadaRoom_KouplerFiber (EK1521)^SBR_2 (EK1501)^Term 77 (EL2809)^Channel 5^Output} *)
	STP.XV204B_AirBlowerValveR4_OpenCmd AT %QX31.5 : BOOL;	(*  ~ {LinkedWith:TIID^C6920 (EtherCAT)^ScadaRoom_KouplerUTP (EK1100)^ScadaRoom_KouplerFiber (EK1521)^SBR_2 (EK1501)^Term 77 (EL2809)^Channel 8^Output} *)
	STP.XV203B_AirBlowerValveR3_OpenCmd AT %QX31.4 : BOOL;	(*  ~ {LinkedWith:TIID^C6920 (EtherCAT)^ScadaRoom_KouplerUTP (EK1100)^ScadaRoom_KouplerFiber (EK1521)^SBR_2 (EK1501)^Term 77 (EL2809)^Channel 7^Output} *)
	STP.XV221B_LimeValveR1_OpenCmd AT %QX31.6 : BOOL;	(*  ~ {LinkedWith:TIID^C6920 (EtherCAT)^ScadaRoom_KouplerUTP (EK1100)^ScadaRoom_KouplerFiber (EK1521)^SBR_2 (EK1501)^Term 77 (EL2809)^Channel 9^Output} *)
	STP.XV222B_LimeValveR2_OpenCmd AT %QX31.7 : BOOL;	(*  ~ {LinkedWith:TIID^C6920 (EtherCAT)^ScadaRoom_KouplerUTP (EK1100)^ScadaRoom_KouplerFiber (EK1521)^SBR_2 (EK1501)^Term 77 (EL2809)^Channel 10^Output} *)
	STP.XV223B_LimeValveR3_OpenCmd AT %QX32.0 : BOOL;	(*  ~ {LinkedWith:TIID^C6920 (EtherCAT)^ScadaRoom_KouplerUTP (EK1100)^ScadaRoom_KouplerFiber (EK1521)^SBR_2 (EK1501)^Term 77 (EL2809)^Channel 11^Output} *)
	STP.XV224B_LimeValveR4_OpenCmd AT %QX32.1 : BOOL;	(*  ~ {LinkedWith:TIID^C6920 (EtherCAT)^ScadaRoom_KouplerUTP (EK1100)^ScadaRoom_KouplerFiber (EK1521)^SBR_2 (EK1501)^Term 77 (EL2809)^Channel 12^Output} *)
	STP.XV211B_AlumValveR1_OpenCmd AT %QX32.2 : BOOL;	(*  ~ {LinkedWith:TIID^C6920 (EtherCAT)^ScadaRoom_KouplerUTP (EK1100)^ScadaRoom_KouplerFiber (EK1521)^SBR_2 (EK1501)^Term 77 (EL2809)^Channel 13^Output} *)
	STP.XV212B_AlumValveR2_OpenCmd AT %QX32.3 : BOOL;	(*  ~ {LinkedWith:TIID^C6920 (EtherCAT)^ScadaRoom_KouplerUTP (EK1100)^ScadaRoom_KouplerFiber (EK1521)^SBR_2 (EK1501)^Term 77 (EL2809)^Channel 14^Output} *)
	STP.XV213B_AlumValveR3_OpenCmd AT %QX32.4 : BOOL;	(*  ~ {LinkedWith:TIID^C6920 (EtherCAT)^ScadaRoom_KouplerUTP (EK1100)^ScadaRoom_KouplerFiber (EK1521)^SBR_2 (EK1501)^Term 77 (EL2809)^Channel 15^Output} *)
	STP.XV214B_AlumValveR4_OpenCmd AT %QX32.5 : BOOL;	(*  ~ {LinkedWith:TIID^C6920 (EtherCAT)^ScadaRoom_KouplerUTP (EK1100)^ScadaRoom_KouplerFiber (EK1521)^SBR_2 (EK1501)^Term 77 (EL2809)^Channel 16^Output} *)
	STP.XV241B_SludgeValveR1_OpenCmd AT %QX32.6 : BOOL;	(*  ~ {LinkedWith:TIID^C6920 (EtherCAT)^ScadaRoom_KouplerUTP (EK1100)^ScadaRoom_KouplerFiber (EK1521)^SBR_2 (EK1501)^Term 78 (EL2809)^Channel 1^Output} *)
	STP.XV242B_SludgeValveR2_OpenCmd AT %QX32.7 : BOOL;	(*  ~ {LinkedWith:TIID^C6920 (EtherCAT)^ScadaRoom_KouplerUTP (EK1100)^ScadaRoom_KouplerFiber (EK1521)^SBR_2 (EK1501)^Term 78 (EL2809)^Channel 2^Output} *)
	STP.XV243B_SludgeValveR3_OpenCmd AT %QX33.0 : BOOL;	(*  ~ {LinkedWith:TIID^C6920 (EtherCAT)^ScadaRoom_KouplerUTP (EK1100)^ScadaRoom_KouplerFiber (EK1521)^SBR_2 (EK1501)^Term 78 (EL2809)^Channel 3^Output} *)
	STP.XV244B_SludgeValveR4_OpenCmd AT %QX33.1 : BOOL;	(*  ~ {LinkedWith:TIID^C6920 (EtherCAT)^ScadaRoom_KouplerUTP (EK1100)^ScadaRoom_KouplerFiber (EK1521)^SBR_2 (EK1501)^Term 78 (EL2809)^Channel 4^Output} *)
	STP.XV241B_SludgeValveR1_CloseCmd AT %QX33.2 : BOOL;	(*  ~ {LinkedWith:TIID^C6920 (EtherCAT)^ScadaRoom_KouplerUTP (EK1100)^ScadaRoom_KouplerFiber (EK1521)^SBR_2 (EK1501)^Term 78 (EL2809)^Channel 5^Output} *)
	STP.XV242B_SludgeValveR2_CloseCmd AT %QX33.3 : BOOL;	(*  ~ {LinkedWith:TIID^C6920 (EtherCAT)^ScadaRoom_KouplerUTP (EK1100)^ScadaRoom_KouplerFiber (EK1521)^SBR_2 (EK1501)^Term 78 (EL2809)^Channel 6^Output} *)
	STP.XV243B_SludgeValveClosedR3_CloseCmd AT %QX33.4 : BOOL;	(*  ~ {LinkedWith:TIID^C6920 (EtherCAT)^ScadaRoom_KouplerUTP (EK1100)^ScadaRoom_KouplerFiber (EK1521)^SBR_2 (EK1501)^Term 78 (EL2809)^Channel 7^Output} *)
	STP.XV244B_SludgeValveR4_CloseCmd AT %QX33.5 : BOOL;	(*  ~ {LinkedWith:TIID^C6920 (EtherCAT)^ScadaRoom_KouplerUTP (EK1100)^ScadaRoom_KouplerFiber (EK1521)^SBR_2 (EK1501)^Term 78 (EL2809)^Channel 8^Output} *)
	STP.XV205B_SBRValveR1_CloseCmd AT %QX33.6 : BOOL;	(*  ~ {LinkedWith:TIID^C6920 (EtherCAT)^ScadaRoom_KouplerUTP (EK1100)^ScadaRoom_KouplerFiber (EK1521)^SBR_2 (EK1501)^Term 79 (EL2809)^Channel 1^Output} *)
	STP.XV206B_SBRValveR2_CloseCmd AT %QX33.7 : BOOL;	(*  ~ {LinkedWith:TIID^C6920 (EtherCAT)^ScadaRoom_KouplerUTP (EK1100)^ScadaRoom_KouplerFiber (EK1521)^SBR_2 (EK1501)^Term 79 (EL2809)^Channel 2^Output} *)
	STP.XV207B_SBRValveR3_CloseCmd AT %QX34.0 : BOOL;	(*  ~ {LinkedWith:TIID^C6920 (EtherCAT)^ScadaRoom_KouplerUTP (EK1100)^ScadaRoom_KouplerFiber (EK1521)^SBR_2 (EK1501)^Term 79 (EL2809)^Channel 3^Output} *)
	STP.XV208B_SBRValveR4_CloseCmd AT %QX34.1 : BOOL;	(*  ~ {LinkedWith:TIID^C6920 (EtherCAT)^ScadaRoom_KouplerUTP (EK1100)^ScadaRoom_KouplerFiber (EK1521)^SBR_2 (EK1501)^Term 79 (EL2809)^Channel 4^Output} *)
	STP.XV201B_AirBlowerValveR1_CloseCmd AT %QX34.2 : BOOL;	(*  ~ {LinkedWith:TIID^C6920 (EtherCAT)^ScadaRoom_KouplerUTP (EK1100)^ScadaRoom_KouplerFiber (EK1521)^SBR_2 (EK1501)^Term 79 (EL2809)^Channel 5^Output} *)
	STP.XV202B_AirBlowerValveR2_CloseCmd AT %QX34.3 : BOOL;	(*  ~ {LinkedWith:TIID^C6920 (EtherCAT)^ScadaRoom_KouplerUTP (EK1100)^ScadaRoom_KouplerFiber (EK1521)^SBR_2 (EK1501)^Term 79 (EL2809)^Channel 6^Output} *)
	STP.XV203B_AirBlowerValveR3_CloseCmd AT %QX34.4 : BOOL;	(*  ~ {LinkedWith:TIID^C6920 (EtherCAT)^ScadaRoom_KouplerUTP (EK1100)^ScadaRoom_KouplerFiber (EK1521)^SBR_2 (EK1501)^Term 79 (EL2809)^Channel 7^Output} *)
	STP.XV204B_AirBlowerValveR4_CloseCmd AT %QX34.5 : BOOL;	(*  ~ {LinkedWith:TIID^C6920 (EtherCAT)^ScadaRoom_KouplerUTP (EK1100)^ScadaRoom_KouplerFiber (EK1521)^SBR_2 (EK1501)^Term 79 (EL2809)^Channel 8^Output} *)
	STP.XV221B_LimeValveR1_CloseCmd AT %QX34.6 : BOOL;	(*  ~ {LinkedWith:TIID^C6920 (EtherCAT)^ScadaRoom_KouplerUTP (EK1100)^ScadaRoom_KouplerFiber (EK1521)^SBR_2 (EK1501)^Term 79 (EL2809)^Channel 9^Output} *)
	STP.XV222B_LimeValveR2_CloseCmd AT %QX34.7 : BOOL;	(*  ~ {LinkedWith:TIID^C6920 (EtherCAT)^ScadaRoom_KouplerUTP (EK1100)^ScadaRoom_KouplerFiber (EK1521)^SBR_2 (EK1501)^Term 79 (EL2809)^Channel 10^Output} *)
	STP.XV223B_LimeValveR3_CloseCmd AT %QX35.0 : BOOL;	(*  ~ {LinkedWith:TIID^C6920 (EtherCAT)^ScadaRoom_KouplerUTP (EK1100)^ScadaRoom_KouplerFiber (EK1521)^SBR_2 (EK1501)^Term 79 (EL2809)^Channel 11^Output} *)
	STP.XV224B_LimeValveR4_CloseCmd AT %QX35.1 : BOOL;	(*  ~ {LinkedWith:TIID^C6920 (EtherCAT)^ScadaRoom_KouplerUTP (EK1100)^ScadaRoom_KouplerFiber (EK1521)^SBR_2 (EK1501)^Term 79 (EL2809)^Channel 12^Output} *)
	STP.XV211B_AlumValveR1_CloseCmd AT %QX35.2 : BOOL;	(*  ~ {LinkedWith:TIID^C6920 (EtherCAT)^ScadaRoom_KouplerUTP (EK1100)^ScadaRoom_KouplerFiber (EK1521)^SBR_2 (EK1501)^Term 79 (EL2809)^Channel 13^Output} *)
	STP.XV212B_AlumValveR2_CloseCmd AT %QX35.3 : BOOL;	(*  ~ {LinkedWith:TIID^C6920 (EtherCAT)^ScadaRoom_KouplerUTP (EK1100)^ScadaRoom_KouplerFiber (EK1521)^SBR_2 (EK1501)^Term 79 (EL2809)^Channel 14^Output} *)
	STP.XV213B_AlumValveR3_CloseCmd AT %QX35.4 : BOOL;	(*  ~ {LinkedWith:TIID^C6920 (EtherCAT)^ScadaRoom_KouplerUTP (EK1100)^ScadaRoom_KouplerFiber (EK1521)^SBR_2 (EK1501)^Term 79 (EL2809)^Channel 15^Output} *)
	STP.XV214B_AlumValveR4_CloseCmd AT %QX35.5 : BOOL;	(*  ~ {LinkedWith:TIID^C6920 (EtherCAT)^ScadaRoom_KouplerUTP (EK1100)^ScadaRoom_KouplerFiber (EK1521)^SBR_2 (EK1501)^Term 79 (EL2809)^Channel 16^Output} *)
	STP.OPR1BON_ReactorR1_OnlineCmd AT %QX35.6 : BOOL;	(*  ~ {LinkedWith:TIID^C6920 (EtherCAT)^ScadaRoom_KouplerUTP (EK1100)^ScadaRoom_KouplerFiber (EK1521)^SBR_2 (EK1501)^Term 80 (EL2809)^Channel 1^Output} *)
	STP.OPR2BON_ReactorR2_OnlineCmd AT %QX35.7 : BOOL;	(*  ~ {LinkedWith:TIID^C6920 (EtherCAT)^ScadaRoom_KouplerUTP (EK1100)^ScadaRoom_KouplerFiber (EK1521)^SBR_2 (EK1501)^Term 80 (EL2809)^Channel 2^Output} *)
	STP.OPR3BON_ReactorR3_OnlineCmd AT %QX36.0 : BOOL;	(*  ~ {LinkedWith:TIID^C6920 (EtherCAT)^ScadaRoom_KouplerUTP (EK1100)^ScadaRoom_KouplerFiber (EK1521)^SBR_2 (EK1501)^Term 80 (EL2809)^Channel 3^Output} *)
	STP.OPR4BON_ReactorR4_OnlineCmd AT %QX36.1 : BOOL;	(*  ~ {LinkedWith:TIID^C6920 (EtherCAT)^ScadaRoom_KouplerUTP (EK1100)^ScadaRoom_KouplerFiber (EK1521)^SBR_2 (EK1501)^Term 80 (EL2809)^Channel 4^Output} *)
	STP.OPR1BOFF_ReactorR1_OfflineCmd AT %QX36.2 : BOOL;	(*  ~ {LinkedWith:TIID^C6920 (EtherCAT)^ScadaRoom_KouplerUTP (EK1100)^ScadaRoom_KouplerFiber (EK1521)^SBR_2 (EK1501)^Term 80 (EL2809)^Channel 5^Output} *)
	STP.OPR2BOFF_ReactorR2_OfflineCmd AT %QX36.3 : BOOL;	(*  ~ {LinkedWith:TIID^C6920 (EtherCAT)^ScadaRoom_KouplerUTP (EK1100)^ScadaRoom_KouplerFiber (EK1521)^SBR_2 (EK1501)^Term 80 (EL2809)^Channel 6^Output} *)
	STP.OPR3BOFF_ReactorR3_OfflineCmd AT %QX36.4 : BOOL;	(*  ~ {LinkedWith:TIID^C6920 (EtherCAT)^ScadaRoom_KouplerUTP (EK1100)^ScadaRoom_KouplerFiber (EK1521)^SBR_2 (EK1501)^Term 80 (EL2809)^Channel 7^Output} *)
	STP.OPR4BOFF_ReactorR4_OfflineCmd AT %QX36.5 : BOOL;	(*  ~ {LinkedWith:TIID^C6920 (EtherCAT)^ScadaRoom_KouplerUTP (EK1100)^ScadaRoom_KouplerFiber (EK1521)^SBR_2 (EK1501)^Term 80 (EL2809)^Channel 8^Output} *)
	STP.OPR1BSW_ReactorR1_SwitchCmd AT %QX36.6 : BOOL;	(*  ~ {LinkedWith:TIID^C6920 (EtherCAT)^ScadaRoom_KouplerUTP (EK1100)^ScadaRoom_KouplerFiber (EK1521)^SBR_2 (EK1501)^Term 81 (EL2809)^Channel 1^Output} *)
	STP.OPR2BSW_ReactorR2_SwitchCmd AT %QX36.7 : BOOL;	(*  ~ {LinkedWith:TIID^C6920 (EtherCAT)^ScadaRoom_KouplerUTP (EK1100)^ScadaRoom_KouplerFiber (EK1521)^SBR_2 (EK1501)^Term 81 (EL2809)^Channel 2^Output} *)
	STP.OPR3BSW_ReactorR3_SwitchCmd AT %QX37.0 : BOOL;	(*  ~ {LinkedWith:TIID^C6920 (EtherCAT)^ScadaRoom_KouplerUTP (EK1100)^ScadaRoom_KouplerFiber (EK1521)^SBR_2 (EK1501)^Term 81 (EL2809)^Channel 3^Output} *)
	STP.OPR4BSW_ReactorR4_SwitchCmd AT %QX37.1 : BOOL;	(*  ~ {LinkedWith:TIID^C6920 (EtherCAT)^ScadaRoom_KouplerUTP (EK1100)^ScadaRoom_KouplerFiber (EK1521)^SBR_2 (EK1501)^Term 81 (EL2809)^Channel 4^Output} *)
	STP.AUX502_PLCRunStat AT %QX72.7 : BOOL;	(*  ~ {LinkedWith:TIID^C6920 (EtherCAT)^ScadaRoom_KouplerUTP (EK1100)^ScadaRoom_KouplerFiber (EK1521)^SBR_2 (EK1501)^Term 81 (EL2809)^Channel 5^Output} *)
	STP.AUX501_CommonAlarm AT %QX73.0 : BOOL;	(*  ~ {LinkedWith:TIID^C6920 (EtherCAT)^ScadaRoom_KouplerUTP (EK1100)^ScadaRoom_KouplerFiber (EK1521)^SBR_2 (EK1501)^Term 81 (EL2809)^Channel 6^Output} *)
	STP.LSHH210A_LimeTank1 AT %IX84.0 : BOOL;	(*  ~ {LinkedWith:TIID^C6920 (EtherCAT)^ScadaRoom_KouplerUTP (EK1100)^ScadaRoom_KouplerFiber (EK1521)^ChemicalAndTertiary (EK1501)^Term 83 (EL1809)^Channel 1^Input} *)
	STP.LSH210A_LimeTank1 AT %IX84.1 : BOOL;	(*  ~ {LinkedWith:TIID^C6920 (EtherCAT)^ScadaRoom_KouplerUTP (EK1100)^ScadaRoom_KouplerFiber (EK1521)^ChemicalAndTertiary (EK1501)^Term 83 (EL1809)^Channel 2^Input} *)
	STP.LSL210A_LimeTank1 AT %IX84.2 : BOOL;	(*  ~ {LinkedWith:TIID^C6920 (EtherCAT)^ScadaRoom_KouplerUTP (EK1100)^ScadaRoom_KouplerFiber (EK1521)^ChemicalAndTertiary (EK1501)^Term 83 (EL1809)^Channel 3^Input} *)
	STP.LSD210A_LimeTank1 AT %IX257.1 : BOOL;	(*  ~ {LinkedWith:TIID^C6920 (EtherCAT)^ScadaRoom_KouplerUTP (EK1100)^ScadaRoom_KouplerFiber (EK1521)^ChemicalAndTertiary (EK1501)^Term 83 (EL1809)^Channel 4^Input} *)
	STP.LSHH210B_LimeTank2 AT %IX152.0 : BOOL;	(*  ~ {LinkedWith:TIID^C6920 (EtherCAT)^ScadaRoom_KouplerUTP (EK1100)^ScadaRoom_KouplerFiber (EK1521)^ChemicalAndTertiary (EK1501)^Term 83 (EL1809)^Channel 5^Input} *)
	STP.LSH210B_LimeTank2 AT %IX84.5 : BOOL;	(*  ~ {LinkedWith:TIID^C6920 (EtherCAT)^ScadaRoom_KouplerUTP (EK1100)^ScadaRoom_KouplerFiber (EK1521)^ChemicalAndTertiary (EK1501)^Term 83 (EL1809)^Channel 6^Input} *)
	STP.LSL210B_LimeTank2 AT %IX84.6 : BOOL;	(*  ~ {LinkedWith:TIID^C6920 (EtherCAT)^ScadaRoom_KouplerUTP (EK1100)^ScadaRoom_KouplerFiber (EK1521)^ChemicalAndTertiary (EK1501)^Term 83 (EL1809)^Channel 7^Input} *)
	STP.LSD210B_LimeTank2 AT %IX257.2 : BOOL;	(*  ~ {LinkedWith:TIID^C6920 (EtherCAT)^ScadaRoom_KouplerUTP (EK1100)^ScadaRoom_KouplerFiber (EK1521)^ChemicalAndTertiary (EK1501)^Term 83 (EL1809)^Channel 8^Input} *)
	STP.LSHH210C_LimeTank3 AT %IX85.0 : BOOL;	(*  ~ {LinkedWith:TIID^C6920 (EtherCAT)^ScadaRoom_KouplerUTP (EK1100)^ScadaRoom_KouplerFiber (EK1521)^ChemicalAndTertiary (EK1501)^Term 83 (EL1809)^Channel 9^Input} *)
	STP.LSH210C_LimeTank3 AT %IX85.1 : BOOL;	(*  ~ {LinkedWith:TIID^C6920 (EtherCAT)^ScadaRoom_KouplerUTP (EK1100)^ScadaRoom_KouplerFiber (EK1521)^ChemicalAndTertiary (EK1501)^Term 83 (EL1809)^Channel 10^Input} *)
	STP.LSL210C_LimeTank3 AT %IX85.2 : BOOL;	(*  ~ {LinkedWith:TIID^C6920 (EtherCAT)^ScadaRoom_KouplerUTP (EK1100)^ScadaRoom_KouplerFiber (EK1521)^ChemicalAndTertiary (EK1501)^Term 83 (EL1809)^Channel 11^Input} *)
	STP.LSD210C_LimeTank3 AT %IX257.3 : BOOL;	(*  ~ {LinkedWith:TIID^C6920 (EtherCAT)^ScadaRoom_KouplerUTP (EK1100)^ScadaRoom_KouplerFiber (EK1521)^ChemicalAndTertiary (EK1501)^Term 83 (EL1809)^Channel 12^Input} *)
	STP.LSL351A_AlumTank1 AT %IX257.4 : BOOL;	(*  ~ {LinkedWith:TIID^C6920 (EtherCAT)^ScadaRoom_KouplerUTP (EK1100)^ScadaRoom_KouplerFiber (EK1521)^ChemicalAndTertiary (EK1501)^Term 83 (EL1809)^Channel 13^Input} *)
	STP.LSL351B_AlumTank2 AT %IX257.5 : BOOL;	(*  ~ {LinkedWith:TIID^C6920 (EtherCAT)^ScadaRoom_KouplerUTP (EK1100)^ScadaRoom_KouplerFiber (EK1521)^ChemicalAndTertiary (EK1501)^Term 83 (EL1809)^Channel 14^Input} *)
	STP.LSL351C_AlumTank3 AT %IX257.6 : BOOL;	(*  ~ {LinkedWith:TIID^C6920 (EtherCAT)^ScadaRoom_KouplerUTP (EK1100)^ScadaRoom_KouplerFiber (EK1521)^ChemicalAndTertiary (EK1501)^Term 83 (EL1809)^Channel 15^Input} *)
	STP.LSL351D_AlumTank4 AT %IX257.7 : BOOL;	(*  ~ {LinkedWith:TIID^C6920 (EtherCAT)^ScadaRoom_KouplerUTP (EK1100)^ScadaRoom_KouplerFiber (EK1521)^ChemicalAndTertiary (EK1501)^Term 83 (EL1809)^Channel 16^Input} *)
	STP.LSL355A_SodiumHypochloriteTank AT %IX258.0 : BOOL;	(*  ~ {LinkedWith:TIID^C6920 (EtherCAT)^ScadaRoom_KouplerUTP (EK1100)^ScadaRoom_KouplerFiber (EK1521)^ChemicalAndTertiary (EK1501)^Term 84 (EL1809)^Channel 1^Input} *)
	STP.LSL355B_SodiumHypochloriteTank AT %IX258.1 : BOOL;	(*  ~ {LinkedWith:TIID^C6920 (EtherCAT)^ScadaRoom_KouplerUTP (EK1100)^ScadaRoom_KouplerFiber (EK1521)^ChemicalAndTertiary (EK1501)^Term 84 (EL1809)^Channel 2^Input} *)
	STP.LSL355C_SodiumHypochloriteTank AT %IX258.2 : BOOL;	(*  ~ {LinkedWith:TIID^C6920 (EtherCAT)^ScadaRoom_KouplerUTP (EK1100)^ScadaRoom_KouplerFiber (EK1521)^ChemicalAndTertiary (EK1501)^Term 84 (EL1809)^Channel 3^Input} *)
	STP.LSL353A_CausticSodaTank AT %IX258.3 : BOOL;	(*  ~ {LinkedWith:TIID^C6920 (EtherCAT)^ScadaRoom_KouplerUTP (EK1100)^ScadaRoom_KouplerFiber (EK1521)^ChemicalAndTertiary (EK1501)^Term 84 (EL1809)^Channel 4^Input} *)
	STP.LSL353B_CausticSodaTank AT %IX258.4 : BOOL;	(*  ~ {LinkedWith:TIID^C6920 (EtherCAT)^ScadaRoom_KouplerUTP (EK1100)^ScadaRoom_KouplerFiber (EK1521)^ChemicalAndTertiary (EK1501)^Term 84 (EL1809)^Channel 5^Input} *)
	STP.LSHH301_EffluentSump AT %IX86.5 : BOOL;	(*  ~ {LinkedWith:TIID^C6920 (EtherCAT)^ScadaRoom_KouplerUTP (EK1100)^ScadaRoom_KouplerFiber (EK1521)^ChemicalAndTertiary (EK1501)^Term 84 (EL1809)^Channel 6^Input} *)
	STP.LSH301_EffluentSump AT %IX86.6 : BOOL;	(*  ~ {LinkedWith:TIID^C6920 (EtherCAT)^ScadaRoom_KouplerUTP (EK1100)^ScadaRoom_KouplerFiber (EK1521)^ChemicalAndTertiary (EK1501)^Term 84 (EL1809)^Channel 7^Input} *)
	STP.LSL301_EffluentSump AT %IX86.7 : BOOL;	(*  ~ {LinkedWith:TIID^C6920 (EtherCAT)^ScadaRoom_KouplerUTP (EK1100)^ScadaRoom_KouplerFiber (EK1521)^ChemicalAndTertiary (EK1501)^Term 84 (EL1809)^Channel 8^Input} *)
	STP.LSHH302_CollectionSump AT %IX87.0 : BOOL;	(*  ~ {LinkedWith:TIID^C6920 (EtherCAT)^ScadaRoom_KouplerUTP (EK1100)^ScadaRoom_KouplerFiber (EK1521)^ChemicalAndTertiary (EK1501)^Term 84 (EL1809)^Channel 9^Input} *)
	STP.LSH302_CollectionSump AT %IX87.1 : BOOL;	(*  ~ {LinkedWith:TIID^C6920 (EtherCAT)^ScadaRoom_KouplerUTP (EK1100)^ScadaRoom_KouplerFiber (EK1521)^ChemicalAndTertiary (EK1501)^Term 84 (EL1809)^Channel 10^Input} *)
	STP.LSL302_CollectionSump AT %IX87.2 : BOOL;	(*  ~ {LinkedWith:TIID^C6920 (EtherCAT)^ScadaRoom_KouplerUTP (EK1100)^ScadaRoom_KouplerFiber (EK1521)^ChemicalAndTertiary (EK1501)^Term 84 (EL1809)^Channel 11^Input} *)
	STP.LSH308A_ReUseWaterStorageTank1HIGH AT %IX87.3 : BOOL;	(*  ~ {LinkedWith:TIID^C6920 (EtherCAT)^ScadaRoom_KouplerUTP (EK1100)^ScadaRoom_KouplerFiber (EK1521)^ChemicalAndTertiary (EK1501)^Term 84 (EL1809)^Channel 12^Input} *)
	STP.LSH308B_ReUseWaterStorageTank2HIGH AT %IX87.4 : BOOL;	(*  ~ {LinkedWith:TIID^C6920 (EtherCAT)^ScadaRoom_KouplerUTP (EK1100)^ScadaRoom_KouplerFiber (EK1521)^ChemicalAndTertiary (EK1501)^Term 84 (EL1809)^Channel 13^Input} *)
	STP.XV251A_LimeSelectorTank_OpenStat AT %IX108.0 : BOOL;	(*  ~ {LinkedWith:TIID^C6920 (EtherCAT)^ScadaRoom_KouplerUTP (EK1100)^ScadaRoom_KouplerFiber (EK1521)^ChemicalAndTertiary (EK1501)^Term 85 (EL1809)^Channel 1^Input} *)
	STP.XV251B_LimeSelectorTank_OpenStat AT %IX108.1 : BOOL;	(*  ~ {LinkedWith:TIID^C6920 (EtherCAT)^ScadaRoom_KouplerUTP (EK1100)^ScadaRoom_KouplerFiber (EK1521)^ChemicalAndTertiary (EK1501)^Term 85 (EL1809)^Channel 2^Input} *)
	STP.XV251C_LimeSelectorTank_OpenStat AT %IX108.2 : BOOL;	(*  ~ {LinkedWith:TIID^C6920 (EtherCAT)^ScadaRoom_KouplerUTP (EK1100)^ScadaRoom_KouplerFiber (EK1521)^ChemicalAndTertiary (EK1501)^Term 85 (EL1809)^Channel 3^Input} *)
	STP.XV251A_LimeSelectorTank_CloseStat AT %IX108.3 : BOOL;	(*  ~ {LinkedWith:TIID^C6920 (EtherCAT)^ScadaRoom_KouplerUTP (EK1100)^ScadaRoom_KouplerFiber (EK1521)^ChemicalAndTertiary (EK1501)^Term 85 (EL1809)^Channel 4^Input} *)
	STP.XV251B_LimSelectorTank_CloseStat AT %IX108.4 : BOOL;	(*  ~ {LinkedWith:TIID^C6920 (EtherCAT)^ScadaRoom_KouplerUTP (EK1100)^ScadaRoom_KouplerFiber (EK1521)^ChemicalAndTertiary (EK1501)^Term 85 (EL1809)^Channel 5^Input} *)
	STP.XV251C_LimeSelectorTank_CloseStat AT %IX108.5 : BOOL;	(*  ~ {LinkedWith:TIID^C6920 (EtherCAT)^ScadaRoom_KouplerUTP (EK1100)^ScadaRoom_KouplerFiber (EK1521)^ChemicalAndTertiary (EK1501)^Term 85 (EL1809)^Channel 6^Input} *)
	STP.OPAlumA_AlumSelectorTank AT %IX108.6 : BOOL;	(*  ~ {LinkedWith:TIID^C6920 (EtherCAT)^ScadaRoom_KouplerUTP (EK1100)^ScadaRoom_KouplerFiber (EK1521)^ChemicalAndTertiary (EK1501)^Term 85 (EL1809)^Channel 7^Input} *)
	STP.OPAlumB_AlumSelectorTank AT %IX108.7 : BOOL;	(*  ~ {LinkedWith:TIID^C6920 (EtherCAT)^ScadaRoom_KouplerUTP (EK1100)^ScadaRoom_KouplerFiber (EK1521)^ChemicalAndTertiary (EK1501)^Term 85 (EL1809)^Channel 8^Input} *)
	STP.OPAlumC_AlumSelectorTank AT %IX109.0 : BOOL;	(*  ~ {LinkedWith:TIID^C6920 (EtherCAT)^ScadaRoom_KouplerUTP (EK1100)^ScadaRoom_KouplerFiber (EK1521)^ChemicalAndTertiary (EK1501)^Term 85 (EL1809)^Channel 9^Input} *)
	STP.OPAlumD_AlumSelectorTank AT %IX109.1 : BOOL;	(*  ~ {LinkedWith:TIID^C6920 (EtherCAT)^ScadaRoom_KouplerUTP (EK1100)^ScadaRoom_KouplerFiber (EK1521)^ChemicalAndTertiary (EK1501)^Term 85 (EL1809)^Channel 10^Input} *)
	STP.OPCausticA_CausticSodaSelectorTank1 AT %IX109.2 : BOOL;	(*  ~ {LinkedWith:TIID^C6920 (EtherCAT)^ScadaRoom_KouplerUTP (EK1100)^ScadaRoom_KouplerFiber (EK1521)^ChemicalAndTertiary (EK1501)^Term 85 (EL1809)^Channel 11^Input} *)
	STP.OPCausticB_CausticSodaSelectorTank2 AT %IX109.3 : BOOL;	(*  ~ {LinkedWith:TIID^C6920 (EtherCAT)^ScadaRoom_KouplerUTP (EK1100)^ScadaRoom_KouplerFiber (EK1521)^ChemicalAndTertiary (EK1501)^Term 85 (EL1809)^Channel 12^Input} *)
	STP.OPSodiumA_SodiumHypochloriteSelectorTank1 AT %IX109.4 : BOOL;	(*  ~ {LinkedWith:TIID^C6920 (EtherCAT)^ScadaRoom_KouplerUTP (EK1100)^ScadaRoom_KouplerFiber (EK1521)^ChemicalAndTertiary (EK1501)^Term 85 (EL1809)^Channel 13^Input} *)
	STP.OPSodiumB_SodiumHypochloriteSelectorTank2 AT %IX109.5 : BOOL;	(*  ~ {LinkedWith:TIID^C6920 (EtherCAT)^ScadaRoom_KouplerUTP (EK1100)^ScadaRoom_KouplerFiber (EK1521)^ChemicalAndTertiary (EK1501)^Term 85 (EL1809)^Channel 14^Input} *)
	STP.OPSodiumC_SodiumHypochloriteSelectorTank3 AT %IX109.6 : BOOL;	(*  ~ {LinkedWith:TIID^C6920 (EtherCAT)^ScadaRoom_KouplerUTP (EK1100)^ScadaRoom_KouplerFiber (EK1521)^ChemicalAndTertiary (EK1501)^Term 85 (EL1809)^Channel 15^Input} *)
	STP.P210A1_LimePumpS1_RunStat AT %IX109.7 : BOOL;	(*  ~ {LinkedWith:TIID^C6920 (EtherCAT)^ScadaRoom_KouplerUTP (EK1100)^ScadaRoom_KouplerFiber (EK1521)^ChemicalAndTertiary (EK1501)^Term 86 (EL1809)^Channel 1^Input} *)
	STP.P210A2_LimePumpS1S2_RunStat AT %IX110.0 : BOOL;	(*  ~ {LinkedWith:TIID^C6920 (EtherCAT)^ScadaRoom_KouplerUTP (EK1100)^ScadaRoom_KouplerFiber (EK1521)^ChemicalAndTertiary (EK1501)^Term 86 (EL1809)^Channel 2^Input} *)
	STP.P210A3_LimePumpS2_RunStat AT %IX110.1 : BOOL;	(*  ~ {LinkedWith:TIID^C6920 (EtherCAT)^ScadaRoom_KouplerUTP (EK1100)^ScadaRoom_KouplerFiber (EK1521)^ChemicalAndTertiary (EK1501)^Term 86 (EL1809)^Channel 3^Input} *)
	STP.P203A_LimeCirculationPump_RunStat AT %IX99.2 : BOOL;	(*  ~ {LinkedWith:TIID^C6920 (EtherCAT)^ScadaRoom_KouplerUTP (EK1100)^ScadaRoom_KouplerFiber (EK1521)^ChemicalAndTertiary (EK1501)^Term 86 (EL1809)^Channel 4^Input} *)
	STP.P203B_LimeCirculationPump_RunStat AT %IX99.3 : BOOL;	(*  ~ {LinkedWith:TIID^C6920 (EtherCAT)^ScadaRoom_KouplerUTP (EK1100)^ScadaRoom_KouplerFiber (EK1521)^ChemicalAndTertiary (EK1501)^Term 86 (EL1809)^Channel 5^Input} *)
	STP.P211A1_AlumPumpSBRS1_RunStat AT %IX99.4 : BOOL;	(*  ~ {LinkedWith:TIID^C6920 (EtherCAT)^ScadaRoom_KouplerUTP (EK1100)^ScadaRoom_KouplerFiber (EK1521)^ChemicalAndTertiary (EK1501)^Term 86 (EL1809)^Channel 6^Input} *)
	STP.P211A2_AlumPumpSBRS1_RunStat AT %IX99.5 : BOOL;	(*  ~ {LinkedWith:TIID^C6920 (EtherCAT)^ScadaRoom_KouplerUTP (EK1100)^ScadaRoom_KouplerFiber (EK1521)^ChemicalAndTertiary (EK1501)^Term 86 (EL1809)^Channel 7^Input} *)
	STP.P211B1_AlumPump1SBRS2_RunStat AT %IX110.2 : BOOL;	(*  ~ {LinkedWith:TIID^C6920 (EtherCAT)^ScadaRoom_KouplerUTP (EK1100)^ScadaRoom_KouplerFiber (EK1521)^ChemicalAndTertiary (EK1501)^Term 86 (EL1809)^Channel 8^Input} *)
	STP.P211B2_AlumPumpSBRS2_RunStat AT %IX99.7 : BOOL;	(*  ~ {LinkedWith:TIID^C6920 (EtherCAT)^ScadaRoom_KouplerUTP (EK1100)^ScadaRoom_KouplerFiber (EK1521)^ChemicalAndTertiary (EK1501)^Term 86 (EL1809)^Channel 9^Input} *)
	STP.P352A_AlumPumpTertiaryDosing_RunStat AT %IX96.5 : BOOL;	(*  ~ {LinkedWith:TIID^C6920 (EtherCAT)^ScadaRoom_KouplerUTP (EK1100)^ScadaRoom_KouplerFiber (EK1521)^ChemicalAndTertiary (EK1501)^Term 86 (EL1809)^Channel 10^Input} *)
	STP.P352B_AlumPumpTertiaryDosing_RunStat AT %IX96.6 : BOOL;	(*  ~ {LinkedWith:TIID^C6920 (EtherCAT)^ScadaRoom_KouplerUTP (EK1100)^ScadaRoom_KouplerFiber (EK1521)^ChemicalAndTertiary (EK1501)^Term 86 (EL1809)^Channel 11^Input} *)
	STP.XV210A1_LimeValveS1_OpenStat AT %IX90.5 : BOOL;	(*  ~ {LinkedWith:TIID^C6920 (EtherCAT)^ScadaRoom_KouplerUTP (EK1100)^ScadaRoom_KouplerFiber (EK1521)^ChemicalAndTertiary (EK1501)^Term 86 (EL1809)^Channel 12^Input} *)
	STP.XV201A2_LimeValveS2_OpenStat AT %IX90.6 : BOOL;	(*  ~ {LinkedWith:TIID^C6920 (EtherCAT)^ScadaRoom_KouplerUTP (EK1100)^ScadaRoom_KouplerFiber (EK1521)^ChemicalAndTertiary (EK1501)^Term 86 (EL1809)^Channel 13^Input} *)
	STP.XV210A1_LimeValveS1_CloseStat AT %IX90.7 : BOOL;	(*  ~ {LinkedWith:TIID^C6920 (EtherCAT)^ScadaRoom_KouplerUTP (EK1100)^ScadaRoom_KouplerFiber (EK1521)^ChemicalAndTertiary (EK1501)^Term 86 (EL1809)^Channel 14^Input} *)
	STP.XV201A2_LimeValveS2_CloseStat AT %IX91.0 : BOOL;	(*  ~ {LinkedWith:TIID^C6920 (EtherCAT)^ScadaRoom_KouplerUTP (EK1100)^ScadaRoom_KouplerFiber (EK1521)^ChemicalAndTertiary (EK1501)^Term 86 (EL1809)^Channel 15^Input} *)
	STP.P354A_CausticSodaPump_RunStat AT %IX100.2 : BOOL;	(*  ~ {LinkedWith:TIID^C6920 (EtherCAT)^ScadaRoom_KouplerUTP (EK1100)^ScadaRoom_KouplerFiber (EK1521)^ChemicalAndTertiary (EK1501)^Term 87 (EL1809)^Channel 1^Input} *)
	STP.P354B_CausticSodaPump_RunStat AT %IX100.3 : BOOL;	(*  ~ {LinkedWith:TIID^C6920 (EtherCAT)^ScadaRoom_KouplerUTP (EK1100)^ScadaRoom_KouplerFiber (EK1521)^ChemicalAndTertiary (EK1501)^Term 87 (EL1809)^Channel 2^Input} *)
	STP.P356A_SodiumHypochloritePumpChlorinetank_RunStat AT %IX110.3 : BOOL;	(*  ~ {LinkedWith:TIID^C6920 (EtherCAT)^ScadaRoom_KouplerUTP (EK1100)^ScadaRoom_KouplerFiber (EK1521)^ChemicalAndTertiary (EK1501)^Term 87 (EL1809)^Channel 3^Input} *)
	STP.P356B_SodiumHypochloritePumpChlorinetank_RunStat AT %IX110.4 : BOOL;	(*  ~ {LinkedWith:TIID^C6920 (EtherCAT)^ScadaRoom_KouplerUTP (EK1100)^ScadaRoom_KouplerFiber (EK1521)^ChemicalAndTertiary (EK1501)^Term 87 (EL1809)^Channel 4^Input} *)
	STP.P204A_SodiumHypochloritePumpDisinfectionTank_RunStat AT %IX258.5 : BOOL;	(*  ~ {LinkedWith:TIID^C6920 (EtherCAT)^ScadaRoom_KouplerUTP (EK1100)^ScadaRoom_KouplerFiber (EK1521)^ChemicalAndTertiary (EK1501)^Term 87 (EL1809)^Channel 5^Input} *)
	STP.P204B_SodiumHypochloritePumpDisinfectionTank_RunStat AT %IX91.6 : BOOL;	(*  ~ {LinkedWith:TIID^C6920 (EtherCAT)^ScadaRoom_KouplerUTP (EK1100)^ScadaRoom_KouplerFiber (EK1521)^ChemicalAndTertiary (EK1501)^Term 87 (EL1809)^Channel 6^Input} *)
	STP.M210A_LimeStirrer_OverloadStat AT %IX280.0 : BOOL;	(*  ~ {LinkedWith:TIID^C6920 (EtherCAT)^ScadaRoom_KouplerUTP (EK1100)^ScadaRoom_KouplerFiber (EK1521)^ChemicalAndTertiary (EK1501)^Term 87 (EL1809)^Channel 7^Input} *)
	STP.M210B_LimeStirrer_OverloadStat AT %IX280.1 : BOOL;	(*  ~ {LinkedWith:TIID^C6920 (EtherCAT)^ScadaRoom_KouplerUTP (EK1100)^ScadaRoom_KouplerFiber (EK1521)^ChemicalAndTertiary (EK1501)^Term 87 (EL1809)^Channel 8^Input} *)
	STP.M210C_LimeStirrer_OverloadStat AT %IX280.2 : BOOL;	(*  ~ {LinkedWith:TIID^C6920 (EtherCAT)^ScadaRoom_KouplerUTP (EK1100)^ScadaRoom_KouplerFiber (EK1521)^ChemicalAndTertiary (EK1501)^Term 87 (EL1809)^Channel 9^Input} *)
	STP.TMT06_FanStatus AT %IX91.7 : BOOL;	(*  ~ {LinkedWith:TIID^C6920 (EtherCAT)^ScadaRoom_KouplerUTP (EK1100)^ScadaRoom_KouplerFiber (EK1521)^ChemicalAndTertiary (EK1501)^Term 88 (EL1809)^Channel 1^Input} *)
	STP.DP06_DoorPanelStatus AT %IX92.0 : BOOL;	(*  ~ {LinkedWith:TIID^C6920 (EtherCAT)^ScadaRoom_KouplerUTP (EK1100)^ScadaRoom_KouplerFiber (EK1521)^ChemicalAndTertiary (EK1501)^Term 88 (EL1809)^Channel 2^Input} *)
	STP.XV250A_LimeWaterIntakeTank_OpenStat AT %IX92.1 : BOOL;	(*  ~ {LinkedWith:TIID^C6920 (EtherCAT)^ScadaRoom_KouplerUTP (EK1100)^ScadaRoom_KouplerFiber (EK1521)^ChemicalAndTertiary (EK1501)^Term 88 (EL1809)^Channel 3^Input} *)
	STP.XV250B_LimeWaterIntakeTank_OpenStat AT %IX92.2 : BOOL;	(*  ~ {LinkedWith:TIID^C6920 (EtherCAT)^ScadaRoom_KouplerUTP (EK1100)^ScadaRoom_KouplerFiber (EK1521)^ChemicalAndTertiary (EK1501)^Term 88 (EL1809)^Channel 4^Input} *)
	STP.XV250C_LimeWaterIntakeTank_OpenStat AT %IX92.3 : BOOL;	(*  ~ {LinkedWith:TIID^C6920 (EtherCAT)^ScadaRoom_KouplerUTP (EK1100)^ScadaRoom_KouplerFiber (EK1521)^ChemicalAndTertiary (EK1501)^Term 88 (EL1809)^Channel 5^Input} *)
	STP.XV250A_LimeWaterIntakeTank_CloseStat AT %IX92.4 : BOOL;	(*  ~ {LinkedWith:TIID^C6920 (EtherCAT)^ScadaRoom_KouplerUTP (EK1100)^ScadaRoom_KouplerFiber (EK1521)^ChemicalAndTertiary (EK1501)^Term 88 (EL1809)^Channel 6^Input} *)
	STP.XV250B_LimeWaterIntakeTank_CloseStat AT %IX92.5 : BOOL;	(*  ~ {LinkedWith:TIID^C6920 (EtherCAT)^ScadaRoom_KouplerUTP (EK1100)^ScadaRoom_KouplerFiber (EK1521)^ChemicalAndTertiary (EK1501)^Term 88 (EL1809)^Channel 7^Input} *)
	STP.XV250C_LimeWaterIntakeTank_CloseStat AT %IX92.6 : BOOL;	(*  ~ {LinkedWith:TIID^C6920 (EtherCAT)^ScadaRoom_KouplerUTP (EK1100)^ScadaRoom_KouplerFiber (EK1521)^ChemicalAndTertiary (EK1501)^Term 88 (EL1809)^Channel 8^Input} *)
	STP.XV303A_LamellaSludgeDischarge_OpenStat AT %IX92.7 : BOOL;	(*  ~ {LinkedWith:TIID^C6920 (EtherCAT)^ScadaRoom_KouplerUTP (EK1100)^ScadaRoom_KouplerFiber (EK1521)^ChemicalAndTertiary (EK1501)^Term 88 (EL1809)^Channel 9^Input} *)
	STP.XV303B_LamellaSludgeDischarge_OpenStat AT %IX93.0 : BOOL;	(*  ~ {LinkedWith:TIID^C6920 (EtherCAT)^ScadaRoom_KouplerUTP (EK1100)^ScadaRoom_KouplerFiber (EK1521)^ChemicalAndTertiary (EK1501)^Term 88 (EL1809)^Channel 10^Input} *)
	STP.XV303C_LamellaSludgeDischarge_OpenStat AT %IX93.1 : BOOL;	(*  ~ {LinkedWith:TIID^C6920 (EtherCAT)^ScadaRoom_KouplerUTP (EK1100)^ScadaRoom_KouplerFiber (EK1521)^ChemicalAndTertiary (EK1501)^Term 88 (EL1809)^Channel 11^Input} *)
	STP.XV303D_LamellaSludgeDischarge_OpenStat AT %IX93.2 : BOOL;	(*  ~ {LinkedWith:TIID^C6920 (EtherCAT)^ScadaRoom_KouplerUTP (EK1100)^ScadaRoom_KouplerFiber (EK1521)^ChemicalAndTertiary (EK1501)^Term 88 (EL1809)^Channel 12^Input} *)
	STP.XV305_TertiaryTreatmentMainValve_OpenStat AT %IX93.3 : BOOL;	(*  ~ {LinkedWith:TIID^C6920 (EtherCAT)^ScadaRoom_KouplerUTP (EK1100)^ScadaRoom_KouplerFiber (EK1521)^ChemicalAndTertiary (EK1501)^Term 88 (EL1809)^Channel 13^Input} *)
	STP.XV303A_LamellaSludgeDischarge_CloseStat AT %IX93.4 : BOOL;	(*  ~ {LinkedWith:TIID^C6920 (EtherCAT)^ScadaRoom_KouplerUTP (EK1100)^ScadaRoom_KouplerFiber (EK1521)^ChemicalAndTertiary (EK1501)^Term 89 (EL1809)^Channel 1^Input} *)
	STP.XV303B_LamellaSludgeDischarge_CloseStat AT %IX93.5 : BOOL;	(*  ~ {LinkedWith:TIID^C6920 (EtherCAT)^ScadaRoom_KouplerUTP (EK1100)^ScadaRoom_KouplerFiber (EK1521)^ChemicalAndTertiary (EK1501)^Term 89 (EL1809)^Channel 2^Input} *)
	STP.XV303C_LamellaSludgeDischarge_CloseStat AT %IX93.6 : BOOL;	(*  ~ {LinkedWith:TIID^C6920 (EtherCAT)^ScadaRoom_KouplerUTP (EK1100)^ScadaRoom_KouplerFiber (EK1521)^ChemicalAndTertiary (EK1501)^Term 89 (EL1809)^Channel 3^Input} *)
	STP.XV303D_LamellaSludgeDischarge_CloseStat AT %IX93.7 : BOOL;	(*  ~ {LinkedWith:TIID^C6920 (EtherCAT)^ScadaRoom_KouplerUTP (EK1100)^ScadaRoom_KouplerFiber (EK1521)^ChemicalAndTertiary (EK1501)^Term 89 (EL1809)^Channel 4^Input} *)
	STP.XV305_TertiaryTreatmentMainValve_CloseStat AT %IX94.0 : BOOL;	(*  ~ {LinkedWith:TIID^C6920 (EtherCAT)^ScadaRoom_KouplerUTP (EK1100)^ScadaRoom_KouplerFiber (EK1521)^ChemicalAndTertiary (EK1501)^Term 89 (EL1809)^Channel 5^Input} *)
	STP.M210A_LimeStirrer_RunStat AT %IX284.0 : BOOL;	(*  ~ {LinkedWith:TIID^C6920 (EtherCAT)^ScadaRoom_KouplerUTP (EK1100)^ScadaRoom_KouplerFiber (EK1521)^ChemicalAndTertiary (EK1501)^Term 88 (EL1809)^Channel 14^Input} *)
	STP.M210B_LimeStirrer_RunStat AT %IX284.1 : BOOL;	(*  ~ {LinkedWith:TIID^C6920 (EtherCAT)^ScadaRoom_KouplerUTP (EK1100)^ScadaRoom_KouplerFiber (EK1521)^ChemicalAndTertiary (EK1501)^Term 88 (EL1809)^Channel 15^Input} *)
	STP.M210C_LimeStirrer_RunStat AT %IX284.2 : BOOL;	(*  ~ {LinkedWith:TIID^C6920 (EtherCAT)^ScadaRoom_KouplerUTP (EK1100)^ScadaRoom_KouplerFiber (EK1521)^ChemicalAndTertiary (EK1501)^Term 88 (EL1809)^Channel 16^Input} *)
	STP.M303A_Floculator_RunStat AT %IX98.3 : BOOL;	(*  ~ {LinkedWith:TIID^C6920 (EtherCAT)^ScadaRoom_KouplerUTP (EK1100)^ScadaRoom_KouplerFiber (EK1521)^ChemicalAndTertiary (EK1501)^Term 89 (EL1809)^Channel 6^Input} *)
	STP.M303B_Floculator_RunStat AT %IX98.4 : BOOL;	(*  ~ {LinkedWith:TIID^C6920 (EtherCAT)^ScadaRoom_KouplerUTP (EK1100)^ScadaRoom_KouplerFiber (EK1521)^ChemicalAndTertiary (EK1501)^Term 89 (EL1809)^Channel 7^Input} *)
	STP.M303C_Floculator_RunStat AT %IX110.5 : BOOL;	(*  ~ {LinkedWith:TIID^C6920 (EtherCAT)^ScadaRoom_KouplerUTP (EK1100)^ScadaRoom_KouplerFiber (EK1521)^ChemicalAndTertiary (EK1501)^Term 89 (EL1809)^Channel 8^Input} *)
	STP.M303D_Floculator_RunStat AT %IX98.6 : BOOL;	(*  ~ {LinkedWith:TIID^C6920 (EtherCAT)^ScadaRoom_KouplerUTP (EK1100)^ScadaRoom_KouplerFiber (EK1521)^ChemicalAndTertiary (EK1501)^Term 89 (EL1809)^Channel 9^Input} *)
	STP.P301A_EffluentTransferPump_RunStat AT %IX101.0 : BOOL;	(*  ~ {LinkedWith:TIID^C6920 (EtherCAT)^ScadaRoom_KouplerUTP (EK1100)^ScadaRoom_KouplerFiber (EK1521)^ChemicalAndTertiary (EK1501)^Term 89 (EL1809)^Channel 10^Input} *)
	STP.P301B_EffluentTransferPump_RunStat AT %IX101.1 : BOOL;	(*  ~ {LinkedWith:TIID^C6920 (EtherCAT)^ScadaRoom_KouplerUTP (EK1100)^ScadaRoom_KouplerFiber (EK1521)^ChemicalAndTertiary (EK1501)^Term 89 (EL1809)^Channel 11^Input} *)
	STP.P302A_CollectionPump_RunStat AT %IX258.6 : BOOL;	(*  ~ {LinkedWith:TIID^C6920 (EtherCAT)^ScadaRoom_KouplerUTP (EK1100)^ScadaRoom_KouplerFiber (EK1521)^ChemicalAndTertiary (EK1501)^Term 89 (EL1809)^Channel 12^Input} *)
	STP.P302B_CollectionPump_RunStat AT %IX101.3 : BOOL;	(*  ~ {LinkedWith:TIID^C6920 (EtherCAT)^ScadaRoom_KouplerUTP (EK1100)^ScadaRoom_KouplerFiber (EK1521)^ChemicalAndTertiary (EK1501)^Term 89 (EL1809)^Channel 13^Input} *)
	STP.K301A_AirCompressor_RunStat AT %IX101.4 : BOOL;	(*  ~ {LinkedWith:TIID^C6920 (EtherCAT)^ScadaRoom_KouplerUTP (EK1100)^ScadaRoom_KouplerFiber (EK1521)^ChemicalAndTertiary (EK1501)^Term 89 (EL1809)^Channel 14^Input} *)
	STP.K301B_AirCompressor_RunStat AT %IX101.5 : BOOL;	(*  ~ {LinkedWith:TIID^C6920 (EtherCAT)^ScadaRoom_KouplerUTP (EK1100)^ScadaRoom_KouplerFiber (EK1521)^ChemicalAndTertiary (EK1501)^Term 89 (EL1809)^Channel 15^Input} *)
	STP.P210A1_LimePumpS1_LocalRemoteStat AT %IX258.7 : BOOL;	(*  ~ {LinkedWith:TIID^C6920 (EtherCAT)^ScadaRoom_KouplerUTP (EK1100)^ScadaRoom_KouplerFiber (EK1521)^ChemicalAndTertiary (EK1501)^Term 90 (EL1809)^Channel 1^Input} *)
	STP.P210A2_LimePumpS1_LocalRemoteStat AT %IX259.0 : BOOL;	(*  ~ {LinkedWith:TIID^C6920 (EtherCAT)^ScadaRoom_KouplerUTP (EK1100)^ScadaRoom_KouplerFiber (EK1521)^ChemicalAndTertiary (EK1501)^Term 90 (EL1809)^Channel 2^Input} *)
	STP.P210A3_LimePumpS1_LocalRemoteStat AT %IX259.1 : BOOL;	(*  ~ {LinkedWith:TIID^C6920 (EtherCAT)^ScadaRoom_KouplerUTP (EK1100)^ScadaRoom_KouplerFiber (EK1521)^ChemicalAndTertiary (EK1501)^Term 90 (EL1809)^Channel 3^Input} *)
	STP.P203A_LimeCirculationPump1_LocalRemoteStat AT %IX111.1 : BOOL;	(*  ~ {LinkedWith:TIID^C6920 (EtherCAT)^ScadaRoom_KouplerUTP (EK1100)^ScadaRoom_KouplerFiber (EK1521)^ChemicalAndTertiary (EK1501)^Term 90 (EL1809)^Channel 6^Input} *)
	STP.P203B_LimeCirculationPump2_LocalRemoteStat AT %IX259.2 : BOOL;	(*  ~ {LinkedWith:TIID^C6920 (EtherCAT)^ScadaRoom_KouplerUTP (EK1100)^ScadaRoom_KouplerFiber (EK1521)^ChemicalAndTertiary (EK1501)^Term 90 (EL1809)^Channel 7^Input} *)
	STP.P211A1_AlumPumpSBRS1_LocalRemoteStat AT %IX96.1 : BOOL;	(*  ~ {LinkedWith:TIID^C6920 (EtherCAT)^ScadaRoom_KouplerUTP (EK1100)^ScadaRoom_KouplerFiber (EK1521)^ChemicalAndTertiary (EK1501)^Term 90 (EL1809)^Channel 8^Input} *)
	STP.P211A2_AlumPumpSBRS1_LocalRemoteStat AT %IX96.2 : BOOL;	(*  ~ {LinkedWith:TIID^C6920 (EtherCAT)^ScadaRoom_KouplerUTP (EK1100)^ScadaRoom_KouplerFiber (EK1521)^ChemicalAndTertiary (EK1501)^Term 90 (EL1809)^Channel 9^Input} *)
	STP.P211B1_AlumPumpSBRS2_LocalRemoteStat AT %IX96.3 : BOOL;	(*  ~ {LinkedWith:TIID^C6920 (EtherCAT)^ScadaRoom_KouplerUTP (EK1100)^ScadaRoom_KouplerFiber (EK1521)^ChemicalAndTertiary (EK1501)^Term 90 (EL1809)^Channel 10^Input} *)
	STP.P211B2_AlumPump2SBRS2_LocalRemoteStat AT %IX96.4 : BOOL;	(*  ~ {LinkedWith:TIID^C6920 (EtherCAT)^ScadaRoom_KouplerUTP (EK1100)^ScadaRoom_KouplerFiber (EK1521)^ChemicalAndTertiary (EK1501)^Term 90 (EL1809)^Channel 11^Input} *)
	STP.P352A_AlumPumpTertiaryDosing_LocalRemoteStat AT %IX111.2 : BOOL;	(*  ~ {LinkedWith:TIID^C6920 (EtherCAT)^ScadaRoom_KouplerUTP (EK1100)^ScadaRoom_KouplerFiber (EK1521)^ChemicalAndTertiary (EK1501)^Term 90 (EL1809)^Channel 12^Input} *)
	STP.P352B_AlumPumpTertiaryDosing_LocalRemoteStat AT %IX111.3 : BOOL;	(*  ~ {LinkedWith:TIID^C6920 (EtherCAT)^ScadaRoom_KouplerUTP (EK1100)^ScadaRoom_KouplerFiber (EK1521)^ChemicalAndTertiary (EK1501)^Term 90 (EL1809)^Channel 13^Input} *)
	STP.P354A_CausticSodaPump_LocalRemoteStat AT %IX111.4 : BOOL;	(*  ~ {LinkedWith:TIID^C6920 (EtherCAT)^ScadaRoom_KouplerUTP (EK1100)^ScadaRoom_KouplerFiber (EK1521)^ChemicalAndTertiary (EK1501)^Term 90 (EL1809)^Channel 14^Input} *)
	STP.P354B_CausticSodaPump_LocalRemoteStat AT %IX111.5 : BOOL;	(*  ~ {LinkedWith:TIID^C6920 (EtherCAT)^ScadaRoom_KouplerUTP (EK1100)^ScadaRoom_KouplerFiber (EK1521)^ChemicalAndTertiary (EK1501)^Term 90 (EL1809)^Channel 15^Input} *)
	STP.P356A_SodiumHypochloritePump_LocalRemoteStat AT %IX112.0 : BOOL;	(*  ~ {LinkedWith:TIID^C6920 (EtherCAT)^ScadaRoom_KouplerUTP (EK1100)^ScadaRoom_KouplerFiber (EK1521)^ChemicalAndTertiary (EK1501)^Term 91 (EL1809)^Channel 3^Input} *)
	STP.P356B_SodiumHypochloritePump_LocalRemoteStat AT %IX112.1 : BOOL;	(*  ~ {LinkedWith:TIID^C6920 (EtherCAT)^ScadaRoom_KouplerUTP (EK1100)^ScadaRoom_KouplerFiber (EK1521)^ChemicalAndTertiary (EK1501)^Term 91 (EL1809)^Channel 4^Input} *)
	STP.P301A_EffluentTransferPump_LocalRemoteStat AT %IX112.2 : BOOL;	(*  ~ {LinkedWith:TIID^C6920 (EtherCAT)^ScadaRoom_KouplerUTP (EK1100)^ScadaRoom_KouplerFiber (EK1521)^ChemicalAndTertiary (EK1501)^Term 91 (EL1809)^Channel 5^Input} *)
	STP.P301B_EffluentTransferPump_LocalRemoteStat AT %IX112.3 : BOOL;	(*  ~ {LinkedWith:TIID^C6920 (EtherCAT)^ScadaRoom_KouplerUTP (EK1100)^ScadaRoom_KouplerFiber (EK1521)^ChemicalAndTertiary (EK1501)^Term 91 (EL1809)^Channel 6^Input} *)
	STP.P302A_CollectionPump_LocalRemoteStat AT %IX112.4 : BOOL;	(*  ~ {LinkedWith:TIID^C6920 (EtherCAT)^ScadaRoom_KouplerUTP (EK1100)^ScadaRoom_KouplerFiber (EK1521)^ChemicalAndTertiary (EK1501)^Term 91 (EL1809)^Channel 7^Input} *)
	STP.P302B_CollectionPump_LocalRemoteStat AT %IX112.5 : BOOL;	(*  ~ {LinkedWith:TIID^C6920 (EtherCAT)^ScadaRoom_KouplerUTP (EK1100)^ScadaRoom_KouplerFiber (EK1521)^ChemicalAndTertiary (EK1501)^Term 91 (EL1809)^Channel 8^Input} *)
	STP.K301A_AirCompressor_LocalRemoteStat AT %IX112.6 : BOOL;	(*  ~ {LinkedWith:TIID^C6920 (EtherCAT)^ScadaRoom_KouplerUTP (EK1100)^ScadaRoom_KouplerFiber (EK1521)^ChemicalAndTertiary (EK1501)^Term 91 (EL1809)^Channel 9^Input} *)
	STP.K301B_AirCompressor_LocalRemoteStat AT %IX112.7 : BOOL;	(*  ~ {LinkedWith:TIID^C6920 (EtherCAT)^ScadaRoom_KouplerUTP (EK1100)^ScadaRoom_KouplerFiber (EK1521)^ChemicalAndTertiary (EK1501)^Term 91 (EL1809)^Channel 10^Input} *)
	STP.M210A_LimeStirrer_LocalRemoteStat AT %IX288.0 : BOOL;	(*  ~ {LinkedWith:TIID^C6920 (EtherCAT)^ScadaRoom_KouplerUTP (EK1100)^ScadaRoom_KouplerFiber (EK1521)^ChemicalAndTertiary (EK1501)^Term 91 (EL1809)^Channel 11^Input} *)
	STP.M210B_LimeStirrer_LocalRemoteStat AT %IX288.1 : BOOL;	(*  ~ {LinkedWith:TIID^C6920 (EtherCAT)^ScadaRoom_KouplerUTP (EK1100)^ScadaRoom_KouplerFiber (EK1521)^ChemicalAndTertiary (EK1501)^Term 91 (EL1809)^Channel 12^Input} *)
	STP.M210C_LimeStirrer_LocalRemoteStat AT %IX288.2 : BOOL;	(*  ~ {LinkedWith:TIID^C6920 (EtherCAT)^ScadaRoom_KouplerUTP (EK1100)^ScadaRoom_KouplerFiber (EK1521)^ChemicalAndTertiary (EK1501)^Term 91 (EL1809)^Channel 13^Input} *)
	STP.P210A1_LimePumpS1_TripStat AT %IX113.0 : BOOL;	(*  ~ {LinkedWith:TIID^C6920 (EtherCAT)^ScadaRoom_KouplerUTP (EK1100)^ScadaRoom_KouplerFiber (EK1521)^ChemicalAndTertiary (EK1501)^Term 92 (EL1809)^Channel 1^Input} *)
	STP.P210A2_LimePumpS1_TripStat AT %IX113.1 : BOOL;	(*  ~ {LinkedWith:TIID^C6920 (EtherCAT)^ScadaRoom_KouplerUTP (EK1100)^ScadaRoom_KouplerFiber (EK1521)^ChemicalAndTertiary (EK1501)^Term 92 (EL1809)^Channel 2^Input} *)
	STP.P210A3_LimePumpS1_TripStat AT %IX113.2 : BOOL;	(*  ~ {LinkedWith:TIID^C6920 (EtherCAT)^ScadaRoom_KouplerUTP (EK1100)^ScadaRoom_KouplerFiber (EK1521)^ChemicalAndTertiary (EK1501)^Term 92 (EL1809)^Channel 3^Input} *)
	STP.P203A_LimeCirculationPump_TripStat AT %IX113.3 : BOOL;	(*  ~ {LinkedWith:TIID^C6920 (EtherCAT)^ScadaRoom_KouplerUTP (EK1100)^ScadaRoom_KouplerFiber (EK1521)^ChemicalAndTertiary (EK1501)^Term 92 (EL1809)^Channel 6^Input} *)
	STP.P203B_LimeCirculationPump_TripStat AT %IX113.4 : BOOL;	(*  ~ {LinkedWith:TIID^C6920 (EtherCAT)^ScadaRoom_KouplerUTP (EK1100)^ScadaRoom_KouplerFiber (EK1521)^ChemicalAndTertiary (EK1501)^Term 92 (EL1809)^Channel 7^Input} *)
	STP.P211A1_AlumPumpSBRS1_TripStat AT %IX113.5 : BOOL;	(*  ~ {LinkedWith:TIID^C6920 (EtherCAT)^ScadaRoom_KouplerUTP (EK1100)^ScadaRoom_KouplerFiber (EK1521)^ChemicalAndTertiary (EK1501)^Term 92 (EL1809)^Channel 8^Input} *)
	STP.P211A2_AlumPumpSBRS1_TripStat AT %IX113.6 : BOOL;	(*  ~ {LinkedWith:TIID^C6920 (EtherCAT)^ScadaRoom_KouplerUTP (EK1100)^ScadaRoom_KouplerFiber (EK1521)^ChemicalAndTertiary (EK1501)^Term 92 (EL1809)^Channel 9^Input} *)
	STP.P211B1_AlumPumpSBRS1_TripStat AT %IX113.7 : BOOL;	(*  ~ {LinkedWith:TIID^C6920 (EtherCAT)^ScadaRoom_KouplerUTP (EK1100)^ScadaRoom_KouplerFiber (EK1521)^ChemicalAndTertiary (EK1501)^Term 92 (EL1809)^Channel 10^Input} *)
	STP.P211B2_AlumPumpSBRS2_TripStat AT %IX114.0 : BOOL;	(*  ~ {LinkedWith:TIID^C6920 (EtherCAT)^ScadaRoom_KouplerUTP (EK1100)^ScadaRoom_KouplerFiber (EK1521)^ChemicalAndTertiary (EK1501)^Term 92 (EL1809)^Channel 11^Input} *)
